KUKA KRL program: EPS_2_251524_MH2A_A_20251127083654.src

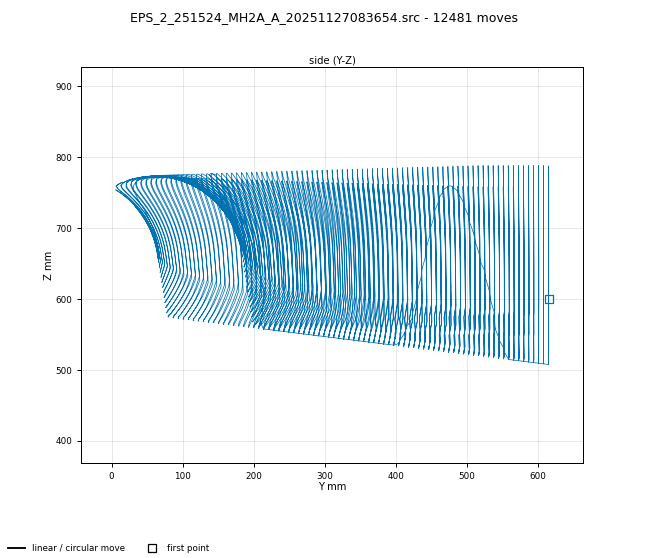
[picture p0: tool path of EPS_2_251524_MH2A_A_20251127083654.src, 12481 of 12483 moves have a stored position in this frame; points joined in program order, loops and branches not executed]
&ACCESS RVP
&REL 4
&COMMENT QRS 19112012
&PARAM EDITMASK = *
DEF PART()
EXT BAS (BAS_COMMAND :IN,REAL :IN )
INT I
BAS (#INITMOV,0 )

;KUKA QRS Post kuka4.cps  Date:22-06-2017 !

File_ID=2930

QRS_PRE_INIT()

;Init var - Until changes are made in qrs_pre_init
Outlet_Square_prg=0
Inlet_1_Square_prg=0
Inlet_2_Square_prg=0
Inlet_3_Square_prg=0
Inlet_4_Square_prg=0
Inlet_5_Square_prg=0

Outlet_1={X 0.000, Y 519.160, Z 687.500, B 0.000, E1 0.000 }
Inlet_1={X 0.000, Y 521.300, Z 657.500, B 0.000, E1 140.000 }
Outlet_1_type=201
Inlet_1_type=201
;QRS#1=Sidecore dimensions
;QRS#2=200-8" PVC SDR 35
;QRS#3=200-8" PVC SDR 35
;QRS#4=
;QRS#5=
;QRS#6=
;QRS#7=
;QRS#8=
;QRS#9=12-08 PSX
;QRS#10=12-08 PSX
;QRS#11=
;QRS#12=
;QRS#13=
;QRS#14=
;QRS#15=
;QRS#16=1220x127x1067 3,5'
;QRS#17=EPS Height
;QRS#18=788
;QRS#19=*
;QRS#20= UPDATED VERSION 22-06-2017
;QRS#21=*
Outlet_Square=0100
Inlet_1_Square=0100
Inlet_2_Square=0
Inlet_3_Square=0
Inlet_4_Square=0
Inlet_5_Square=0
Mill_Square=1
Outlet_Square_Prg=204
Inlet_1_Square_prg=204

QRS_INIT()

$ADVANCE=5

; T1
PTP {E1 173.595,E2 173.595}
PTP {X 0,Y 615.504,A -85,B 0,C 180,E1 173.595,E2 173.595,E3 0,E4 0,E5 0,E6 0}
QRS_SPEED_INIT()
LIN {X 0,Y 615.504,Z 600,A -85,B 0,C 180,E1 173.595,E2 173.595,E3 0,E4 0,E5 0,E6 0} C_VEL
LIN {X 0,Y 615.504,Z 517.862,A -85,B 0,C 180,E1 173.595,E2 173.595} C_VEL
LIN {X 0,Y 615.504,Z 509.682,A -85,B 0,C 180,E1 173.595,E2 173.595} C_VEL
LIN {X 0,Y 615.489,Z 507.682,A -85,B 0,C 180,E1 173.409,E2 173.409} C_VEL
LIN {X 0,Y 615.481,Z 507.697,A -85,B 0,C 180,E1 170.801,E2 170.801} C_VEL
LIN {X 0,Y 615.479,Z 507.69,A -85,B 0,C 180,E1 168.139,E2 168.139} C_VEL
LIN {X 0,Y 615.488,Z 507.682,A -85,B 0,C 180,E1 165.451,E2 165.451} C_VEL
LIN {X 0,Y 615.483,Z 507.699,A -85,B 0,C 180,E1 162.73,E2 162.73} C_VEL
LIN {X 0,Y 615.477,Z 507.687,A -85,B 0,C 180,E1 159.967,E2 159.967} C_VEL
LIN {X 0,Y 615.481,Z 507.683,A -85,B 0,C 180,E1 157.652,E2 157.652} C_VEL
LIN {X 0,Y 615.479,Z 507.692,A -85,B 0,C 180,E1 155.008,E2 155.008} C_VEL
LIN {X 0,Y 615.482,Z 507.688,A -85,B 0,C 180,E1 152.085,E2 152.085} C_VEL
LIN {X 0,Y 615.491,Z 507.714,A -85,B 0,C 180,E1 149.212,E2 149.212} C_VEL
LIN {X 0,Y 615.495,Z 524.435,A -85,B 0,C 180,E1 146.462,E2 146.462} C_VEL
LIN {X 0,Y 615.481,Z 542.244,A -85,B 0,C 180,E1 143.575,E2 143.575} C_VEL
LIN {X 0,Y 615.483,Z 546.958,A -85,B 0,C 180,E1 142.815,E2 142.815} C_VEL
LIN {X 0,Y 615.482,Z 654.02,A -85,B 0,C 180,E1 141.541,E2 141.541} C_VEL
LIN {X 0,Y 615.488,Z 667.054,A -85,B 0,C 180,E1 141.254,E2 141.254} C_VEL
LIN {X 0,Y 615.48,Z 679.367,A -85,B 0,C 180,E1 140.851,E2 140.851} C_VEL
LIN {X 0,Y 615.498,Z 691.041,A -85,B 0,C 180,E1 140.337,E2 140.337} C_VEL
LIN {X 0,Y 615.483,Z 702.98,A -85,B 0,C 180,E1 139.652,E2 139.652} C_VEL
LIN {X 0,Y 615.496,Z 713.375,A -85,B 0,C 180,E1 138.903,E2 138.903} C_VEL
LIN {X 0,Y 615.499,Z 722.741,A -85,B 0,C 180,E1 138.071,E2 138.071} C_VEL
LIN {X 0,Y 615.496,Z 731.335,A -85,B 0,C 180,E1 137.125,E2 137.125} C_VEL
LIN {X 0,Y 615.495,Z 738.265,A -85,B 0,C 180,E1 136.19,E2 136.19} C_VEL
LIN {X 0,Y 615.496,Z 744.904,A -85,B 0,C 180,E1 135.066,E2 135.066} C_VEL
LIN {X 0,Y 615.495,Z 749.711,A -85,B 0,C 180,E1 133.999,E2 133.999} C_VEL
LIN {X 0,Y 615.495,Z 752.959,A -85,B 0,C 180,E1 133.049,E2 133.049} C_VEL
LIN {X 0,Y 615.498,Z 755.309,A -85,B 0,C 180,E1 132.082,E2 132.082} C_VEL
LIN {X 0,Y 615.492,Z 756.779,A -85,B 0,C 180,E1 131.096,E2 131.096} C_VEL
LIN {X 0,Y 615.493,Z 757.346,A -85,B 0,C 180,E1 129.748,E2 129.748} C_VEL
LIN {X 0,Y 615.493,Z 756.882,A -85,B 0,C 180,E1 128.902,E2 128.902} C_VEL
LIN {X 0,Y 615.495,Z 755.644,A -85,B 0,C 180,E1 128.014,E2 128.014} C_VEL
LIN {X 0,Y 615.497,Z 753.167,A -85,B 0,C 180,E1 126.938,E2 126.938} C_VEL
LIN {X 0,Y 615.496,Z 749.426,A -85,B 0,C 180,E1 125.835,E2 125.835} C_VEL
LIN {X 0,Y 615.496,Z 744.143,A -85,B 0,C 180,E1 124.703,E2 124.703} C_VEL
LIN {X 0,Y 615.496,Z 737.021,A -85,B 0,C 180,E1 123.536,E2 123.536} C_VEL
LIN {X 0,Y 615.498,Z 730.229,A -85,B 0,C 180,E1 122.65,E2 122.65} C_VEL
LIN {X 0,Y 615.497,Z 722.8,A -85,B 0,C 180,E1 121.845,E2 121.845} C_VEL
LIN {X 0,Y 615.496,Z 713.317,A -85,B 0,C 180,E1 121.003,E2 121.003} C_VEL
LIN {X 0,Y 615.495,Z 702.902,A -85,B 0,C 180,E1 120.253,E2 120.253} C_VEL
LIN {X 0,Y 615.48,Z 691.58,A -85,B 0,C 180,E1 119.6,E2 119.6} C_VEL
LIN {X 0,Y 615.493,Z 679.846,A -85,B 0,C 180,E1 119.077,E2 119.077} C_VEL
LIN {X 0,Y 615.477,Z 667.095,A -85,B 0,C 180,E1 118.657,E2 118.657} C_VEL
LIN {X 0,Y 615.484,Z 654.766,A -85,B 0,C 180,E1 118.383,E2 118.383} C_VEL
LIN {X 0,Y 615.485,Z 578.99,A -85,B 0,C 180,E1 117.475,E2 117.475} C_VEL
LIN {X 0,Y 615.492,Z 546.957,A -85,B 0,C 180,E1 117.095,E2 117.095} C_VEL
LIN {X 0,Y 615.487,Z 529.495,A -85,B 0,C 180,E1 114.271,E2 114.271} C_VEL
LIN {X 0,Y 615.491,Z 512.144,A -85,B 0,C 180,E1 111.431,E2 111.431} C_VEL
LIN {X 0,Y 615.477,Z 507.687,A -85,B 0,C 180,E1 110.686,E2 110.686} C_VEL
LIN {X 0,Y 615.488,Z 507.683,A -85,B 0,C 180,E1 107.956,E2 107.956} C_VEL
LIN {X 0,Y 615.493,Z 507.701,A -85,B 0,C 180,E1 105.225,E2 105.225} C_VEL
LIN {X 0,Y 615.477,Z 507.686,A -85,B 0,C 180,E1 102.529,E2 102.529} C_VEL
LIN {X 0,Y 615.487,Z 507.684,A -85,B 0,C 180,E1 99.861,E2 99.861} C_VEL
LIN {X 0,Y 615.491,Z 507.7,A -85,B 0,C 180,E1 97.215,E2 97.215} C_VEL
LIN {X 0,Y 615.477,Z 507.688,A -85,B 0,C 180,E1 94.584,E2 94.584} C_VEL
LIN {X 0,Y 615.496,Z 507.68,A -85,B 0,C 180,E1 91.962,E2 91.962} C_VEL
LIN {X 0,Y 615.483,Z 507.694,A -85,B 0,C 180,E1 89.345,E2 89.345} C_VEL
LIN {X 0,Y 615.482,Z 507.693,A -85,B 0,C 180,E1 86.726,E2 86.726} C_VEL
LIN {X 0,Y 615.488,Z 507.681,A -85,B 0,C 180,E1 84.101,E2 84.101} C_VEL
LIN {X 0,Y 615.476,Z 507.69,A -85,B 0,C 180,E1 81.462,E2 81.462} C_VEL
LIN {X 0,Y 615.489,Z 507.696,A -85,B 0,C 180,E1 78.806,E2 78.806} C_VEL
LIN {X 0,Y 615.484,Z 507.682,A -85,B 0,C 180,E1 76.067,E2 76.067} C_VEL
LIN {X 0,Y 615.477,Z 507.689,A -85,B 0,C 180,E1 73.412,E2 73.412} C_VEL
LIN {X 0,Y 615.484,Z 507.695,A -85,B 0,C 180,E1 70.661,E2 70.661} C_VEL
LIN {X 0,Y 615.494,Z 507.68,A -85,B 0,C 180,E1 67.863,E2 67.863} C_VEL
LIN {X 0,Y 615.488,Z 507.696,A -85,B 0,C 180,E1 65.007,E2 65.007} C_VEL
LIN {X 0,Y 615.484,Z 507.684,A -85,B 0,C 180,E1 62.084,E2 62.084} C_VEL
LIN {X 0,Y 615.499,Z 507.679,A -85,B 0,C 180,E1 59.84,E2 59.84} C_VEL
LIN {X 0,Y 615.481,Z 507.684,A -85,B 0,C 180,E1 57.541,E2 57.541} C_VEL
LIN {X 0,Y 615.478,Z 507.69,A -85,B 0,C 180,E1 55.184,E2 55.184} C_VEL
LIN {X 0,Y 615.493,Z 507.699,A -85,B 0,C 180,E1 52.757,E2 52.757} C_VEL
LIN {X 0,Y 615.49,Z 507.682,A -85,B 0,C 180,E1 49.91,E2 49.91} C_VEL
LIN {X 0,Y 615.49,Z 507.681,A -85,B 0,C 180,E1 47.646,E2 47.646} C_VEL
LIN {X 0,Y 615.482,Z 507.693,A -85,B 0,C 180,E1 44.93,E2 44.93} C_VEL
LIN {X 0,Y 615.482,Z 507.688,A -85,B 0,C 180,E1 42.079,E2 42.079} C_VEL
LIN {X 0,Y 615.498,Z 507.68,A -85,B 0,C 180,E1 39.749,E2 39.749} C_VEL
LIN {X 0,Y 615.48,Z 507.691,A -85,B 0,C 180,E1 36.935,E2 36.935} C_VEL
LIN {X 0,Y 615.494,Z 507.695,A -85,B 0,C 180,E1 34.7,E2 34.7} C_VEL
LIN {X 0,Y 615.487,Z 507.682,A -85,B 0,C 180,E1 31.685,E2 31.685} C_VEL
LIN {X 0,Y 615.482,Z 507.683,A -85,B 0,C 180,E1 29.406,E2 29.406} C_VEL
LIN {X 0,Y 615.478,Z 507.687,A -85,B 0,C 180,E1 27.042,E2 27.042} C_VEL
LIN {X 0,Y 615.491,Z 507.696,A -85,B 0,C 180,E1 24.271,E2 24.271} C_VEL
LIN {X 0,Y 615.486,Z 507.682,A -85,B 0,C 180,E1 21.432,E2 21.432} C_VEL
LIN {X 0,Y 615.492,Z 507.693,A -85,B 0,C 180,E1 18.604,E2 18.604} C_VEL
LIN {X 0,Y 615.487,Z 507.689,A -85,B 0,C 180,E1 15.905,E2 15.905} C_VEL
LIN {X 0,Y 615.478,Z 507.684,A -85,B 0,C 180,E1 13.201,E2 13.201} C_VEL
LIN {X 0,Y 615.488,Z 507.693,A -85,B 0,C 180,E1 10.527,E2 10.527} C_VEL
LIN {X 0,Y 615.488,Z 507.69,A -85,B 0,C 180,E1 7.875,E2 7.875} C_VEL
LIN {X 0,Y 615.481,Z 507.683,A -85,B 0,C 180,E1 5.241,E2 5.241} C_VEL
LIN {X 0,Y 615.491,Z 507.688,A -85,B 0,C 180,E1 2.618,E2 2.618} C_VEL
LIN {X 0,Y 615.492,Z 507.695,A -85,B 0,C 180,E1 0,E2 0} C_VEL
LIN {X 0,Y 615.491,Z 507.682,A -85,B 0,C 180,E1 -2.618,E2 -2.618} C_VEL
LIN {X 0,Y 615.481,Z 507.686,A -85,B 0,C 180,E1 -5.242,E2 -5.242} C_VEL
LIN {X 0,Y 615.487,Z 507.702,A -85,B 0,C 180,E1 -7.876,E2 -7.876} C_VEL
LIN {X 0,Y 615.491,Z 507.684,A -85,B 0,C 180,E1 -10.527,E2 -10.527} C_VEL
LIN {X 0,Y 615.478,Z 507.685,A -85,B 0,C 180,E1 -13.202,E2 -13.202} C_VEL
LIN {X 0,Y 615.492,Z 507.699,A -85,B 0,C 180,E1 -15.905,E2 -15.905} C_VEL
LIN {X 0,Y 615.49,Z 507.684,A -85,B 0,C 180,E1 -18.646,E2 -18.646} C_VEL
LIN {X 0,Y 615.486,Z 507.685,A -85,B 0,C 180,E1 -21.432,E2 -21.432} C_VEL
LIN {X 0,Y 615.493,Z 507.694,A -85,B 0,C 180,E1 -24.272,E2 -24.272} C_VEL
LIN {X 0,Y 615.478,Z 507.684,A -85,B 0,C 180,E1 -27.042,E2 -27.042} C_VEL
LIN {X 0,Y 615.488,Z 507.691,A -85,B 0,C 180,E1 -29.794,E2 -29.794} C_VEL
LIN {X 0,Y 615.494,Z 507.691,A -85,B 0,C 180,E1 -32.457,E2 -32.457} C_VEL
LIN {X 0,Y 615.49,Z 507.684,A -85,B 0,C 180,E1 -34.815,E2 -34.815} C_VEL
LIN {X 0,Y 615.474,Z 507.684,A -85,B 0,C 180,E1 -37.243,E2 -37.243} C_VEL
LIN {X 0,Y 615.482,Z 507.698,A -85,B 0,C 180,E1 -40.088,E2 -40.088} C_VEL
LIN {X 0,Y 615.496,Z 507.697,A -85,B 0,C 180,E1 -42.353,E2 -42.353} C_VEL
LIN {X 0,Y 615.48,Z 507.684,A -85,B 0,C 180,E1 -45.07,E2 -45.07} C_VEL
LIN {X 0,Y 615.488,Z 507.689,A -85,B 0,C 180,E1 -47.92,E2 -47.92} C_VEL
LIN {X 0,Y 615.49,Z 507.699,A -85,B 0,C 180,E1 -50.249,E2 -50.249} C_VEL
LIN {X 0,Y 615.482,Z 507.685,A -85,B 0,C 180,E1 -53.065,E2 -53.065} C_VEL
LIN {X 0,Y 615.477,Z 507.684,A -85,B 0,C 180,E1 -55.301,E2 -55.301} C_VEL
LIN {X 0,Y 615.488,Z 507.683,A -85,B 0,C 180,E1 -57.67,E2 -57.67} C_VEL
LIN {X 0,Y 615.495,Z 507.695,A -85,B 0,C 180,E1 -60.593,E2 -60.593} C_VEL
LIN {X 0,Y 615.491,Z 507.686,A -85,B 0,C 180,E1 -62.955,E2 -62.955} C_VEL
LIN {X 0,Y 615.487,Z 507.683,A -85,B 0,C 180,E1 -65.727,E2 -65.727} C_VEL
LIN {X 0,Y 615.492,Z 507.756,A -85,B 0,C 180,E1 -67.837,E2 -67.837} C_VEL
LIN {X 0,Y 615.483,Z 528.07,A -85,B 0,C 180,E1 -70.661,E2 -70.661} C_VEL
LIN {X 0,Y 615.477,Z 548.18,A -85,B 0,C 180,E1 -73.412,E2 -73.412} C_VEL
LIN {X 0,Y 615.487,Z 568.265,A -85,B 0,C 180,E1 -76.125,E2 -76.125} C_VEL
LIN {X 0,Y 615.485,Z 576.034,A -85,B 0,C 180,E1 -77.134,E2 -77.134} C_VEL
LIN {X 0,Y 615.477,Z 683.784,A -85,B 0,C 180,E1 -78.41,E2 -78.41} C_VEL
LIN {X 0,Y 615.482,Z 696.314,A -85,B 0,C 180,E1 -78.681,E2 -78.681} C_VEL
LIN {X 0,Y 615.497,Z 709.493,A -85,B 0,C 180,E1 -79.109,E2 -79.109} C_VEL
LIN {X 0,Y 615.48,Z 721.461,A -85,B 0,C 180,E1 -79.638,E2 -79.638} C_VEL
LIN {X 0,Y 615.481,Z 732.983,A -85,B 0,C 180,E1 -80.303,E2 -80.303} C_VEL
LIN {X 0,Y 615.499,Z 743.33,A -85,B 0,C 180,E1 -81.049,E2 -81.049} C_VEL
LIN {X 0,Y 615.497,Z 751.802,A -85,B 0,C 180,E1 -81.793,E2 -81.793} C_VEL
LIN {X 0,Y 615.498,Z 759.599,A -85,B 0,C 180,E1 -82.619,E2 -82.619} C_VEL
LIN {X 0,Y 615.496,Z 767.197,A -85,B 0,C 180,E1 -83.607,E2 -83.607} C_VEL
LIN {X 0,Y 615.498,Z 774.2,A -85,B 0,C 180,E1 -84.758,E2 -84.758} C_VEL
LIN {X 0,Y 615.493,Z 778.848,A -85,B 0,C 180,E1 -85.743,E2 -85.743} C_VEL
LIN {X 0,Y 615.495,Z 782.396,A -85,B 0,C 180,E1 -86.726,E2 -86.726} C_VEL
LIN {X 0,Y 615.497,Z 784.231,A -85,B 0,C 180,E1 -87.381,E2 -87.381} C_VEL
LIN {X 0,Y 615.496,Z 785.607,A -85,B 0,C 180,E1 -88.036,E2 -88.036} C_VEL
LIN {X 0,Y 615.496,Z 787.173,A -85,B 0,C 180,E1 -89.345,E2 -89.345} C_VEL
LIN {X 0,Y 615.494,Z 787.389,A -85,B 0,C 180,E1 -89.999,E2 -89.999} C_VEL
LIN {X 0,Y 615.496,Z 786.581,A -85,B 0,C 180,E1 -91.308,E2 -91.308} C_VEL
LIN {X 0,Y 615.496,Z 785.61,A -85,B 0,C 180,E1 -91.962,E2 -91.962} C_VEL
LIN {X 0,Y 615.497,Z 784.235,A -85,B 0,C 180,E1 -92.617,E2 -92.617} C_VEL
LIN {X 0,Y 615.496,Z 781.353,A -85,B 0,C 180,E1 -93.6,E2 -93.6} C_VEL
LIN {X 0,Y 615.498,Z 777.446,A -85,B 0,C 180,E1 -94.583,E2 -94.583} C_VEL
LIN {X 0,Y 615.499,Z 772.41,A -85,B 0,C 180,E1 -95.569,E2 -95.569} C_VEL
LIN {X 0,Y 615.496,Z 765.87,A -85,B 0,C 180,E1 -96.583,E2 -96.583} C_VEL
LIN {X 0,Y 615.497,Z 758.142,A -85,B 0,C 180,E1 -97.544,E2 -97.544} C_VEL
LIN {X 0,Y 615.498,Z 750.056,A -85,B 0,C 180,E1 -98.37,E2 -98.37} C_VEL
LIN {X 0,Y 615.499,Z 740.181,A -85,B 0,C 180,E1 -99.198,E2 -99.198} C_VEL
LIN {X 0,Y 615.483,Z 729,A -85,B 0,C 180,E1 -99.944,E2 -99.944} C_VEL
LIN {X 0,Y 615.481,Z 718.045,A -85,B 0,C 180,E1 -100.526,E2 -100.526} C_VEL
LIN {X 0,Y 615.499,Z 705.435,A -85,B 0,C 180,E1 -101.042,E2 -101.042} C_VEL
LIN {X 0,Y 615.479,Z 693.112,A -85,B 0,C 180,E1 -101.401,E2 -101.401} C_VEL
LIN {X 0,Y 615.477,Z 679.544,A -85,B 0,C 180,E1 -101.651,E2 -101.651} C_VEL
LIN {X 0,Y 615.486,Z 575.649,A -85,B 0,C 180,E1 -102.885,E2 -102.885} C_VEL
LIN {X 0,Y 615.479,Z 554.474,A -85,B 0,C 180,E1 -105.734,E2 -105.734} C_VEL
LIN {X 0,Y 615.479,Z 534.611,A -85,B 0,C 180,E1 -108.44,E2 -108.44} C_VEL
LIN {X 0,Y 615.497,Z 514.247,A -85,B 0,C 180,E1 -111.255,E2 -111.255} C_VEL
LIN {X 0,Y 615.489,Z 507.683,A -85,B 0,C 180,E1 -112.187,E2 -112.187} C_VEL
LIN {X 0,Y 615.488,Z 507.687,A -85,B 0,C 180,E1 -114.99,E2 -114.99} C_VEL
LIN {X 0,Y 615.483,Z 507.69,A -85,B 0,C 180,E1 -117.914,E2 -117.914} C_VEL
LIN {X 0,Y 615.499,Z 507.681,A -85,B 0,C 180,E1 -120.158,E2 -120.158} C_VEL
LIN {X 0,Y 615.481,Z 507.683,A -85,B 0,C 180,E1 -122.456,E2 -122.456} C_VEL
LIN {X 0,Y 615.478,Z 507.687,A -85,B 0,C 180,E1 -124.814,E2 -124.814} C_VEL
LIN {X 0,Y 615.496,Z 507.693,A -85,B 0,C 180,E1 -127.24,E2 -127.24} C_VEL
LIN {X 0,Y 615.49,Z 507.684,A -85,B 0,C 180,E1 -130.089,E2 -130.089} C_VEL
LIN {X 0,Y 615.49,Z 507.681,A -85,B 0,C 180,E1 -132.351,E2 -132.351} C_VEL
LIN {X 0,Y 615.481,Z 507.691,A -85,B 0,C 180,E1 -135.067,E2 -135.067} C_VEL
LIN {X 0,Y 615.477,Z 507.69,A -85,B 0,C 180,E1 -137.919,E2 -137.919} C_VEL
LIN {X 0,Y 615.498,Z 507.68,A -85,B 0,C 180,E1 -140.25,E2 -140.25} C_VEL
LIN {X 0,Y 615.48,Z 507.691,A -85,B 0,C 180,E1 -143.062,E2 -143.062} C_VEL
LIN {X 0,Y 615.494,Z 507.696,A -85,B 0,C 180,E1 -145.296,E2 -145.296} C_VEL
LIN {X 0,Y 615.485,Z 507.683,A -85,B 0,C 180,E1 -148.314,E2 -148.314} C_VEL
LIN {X 0,Y 615.482,Z 507.683,A -85,B 0,C 180,E1 -150.593,E2 -150.593} C_VEL
LIN {X 0,Y 615.478,Z 507.69,A -85,B 0,C 180,E1 -152.954,E2 -152.954} C_VEL
LIN {X 0,Y 615.478,Z 507.695,A -85,B 0,C 180,E1 -155.727,E2 -155.727} C_VEL
LIN {X 0,Y 615.486,Z 507.683,A -85,B 0,C 180,E1 -158.568,E2 -158.568} C_VEL
LIN {X 0,Y 615.494,Z 507.7,A -85,B 0,C 180,E1 -161.389,E2 -161.389} C_VEL
LIN {X 0,Y 615.48,Z 507.686,A -85,B 0,C 180,E1 -164.094,E2 -164.094} C_VEL
LIN {X 0,Y 615.478,Z 507.687,A -85,B 0,C 180,E1 -166.798,E2 -166.798} C_VEL
LIN {X 0,Y 615.488,Z 507.701,A -85,B 0,C 180,E1 -169.473,E2 -169.473} C_VEL
LIN {X 0,Y 615.479,Z 507.686,A -85,B 0,C 180,E1 -172.124,E2 -172.124} C_VEL
LIN {X 0,Y 615.481,Z 507.686,A -85,B 0,C 180,E1 -174.758,E2 -174.758} C_VEL
LIN {X 0,Y 615.495,Z 507.7,A -85,B 0,C 180,E1 -177.382,E2 -177.382} C_VEL
LIN {X 0,Y 615.477,Z 507.688,A -85,B 0,C 180,E1 -180,E2 -180} C_VEL
LIN {X 0,Y 615.492,Z 507.682,A -85,B 0,C 180,E1 -182.617,E2 -182.617} C_VEL
LIN {X 0,Y 615.481,Z 507.698,A -85,B 0,C 180,E1 -185.241,E2 -185.241} C_VEL
LIN {X 0,Y 615.489,Z 507.682,A -85,B 0,C 180,E1 -186.591,E2 -186.591} C_VEL
LIN {X 0,Y 614.808,Z 507.844,A -85,B 0,C 180,E1 -187.137,E2 -187.137} C_VEL
LIN {X 0,Y 611.969,Z 508.251,A -85,B 0,C 180,E1 -188.023,E2 -188.023} C_VEL
LIN {X 0,Y 609.577,Z 508.566,A -85,B 0,C 180,E1 -188.735,E2 -188.735} C_VEL
LIN {X 0,Y 608.541,Z 508.686,A -85,B 0,C 180,E1 -189.285,E2 -189.285} C_VEL
LIN {X 0,Y 608.452,Z 508.694,A -85,B 0,C 180,E1 -189.471,E2 -189.471} C_VEL
LIN {X 0,Y 608.456,Z 508.688,A -85,B 0,C 180,E1 -192,E2 -192} C_VEL
LIN {X 0,Y 608.473,Z 508.686,A -85,B 0,C 180,E1 -194.72,E2 -194.72} C_VEL
LIN {X 0,Y 608.447,Z 508.698,A -85,B 0,C 180,E1 -197.476,E2 -197.476} C_VEL
LIN {X 0,Y 608.457,Z 508.687,A -85,B 0,C 180,E1 -200.274,E2 -200.274} C_VEL
LIN {X 0,Y 608.449,Z 508.688,A -85,B 0,C 180,E1 -202.478,E2 -202.478} C_VEL
LIN {X 0,Y 608.451,Z 508.697,A -85,B 0,C 180,E1 -205.301,E2 -205.301} C_VEL
LIN {X 0,Y 608.444,Z 508.697,A -85,B 0,C 180,E1 -207.518,E2 -207.518} C_VEL
LIN {X 0,Y 608.451,Z 508.69,A -85,B 0,C 180,E1 -209.972,E2 -209.972} C_VEL
LIN {X 0,Y 608.513,Z 508.816,A -85,B 0,C 180,E1 -210.734,E2 -210.734} C_VEL
LIN {X 0,Y 608.493,Z 526.519,A -85,B 0,C 180,E1 -213.668,E2 -213.668} C_VEL
LIN {X 0,Y 608.482,Z 543.856,A -85,B 0,C 180,E1 -216.5,E2 -216.5} C_VEL
LIN {X 0,Y 608.461,Z 547.129,A -85,B 0,C 180,E1 -217.03,E2 -217.03} C_VEL
LIN {X 0,Y 608.555,Z 654.443,A -85,B 0,C 180,E1 -218.331,E2 -218.331} C_VEL
LIN {X 0,Y 608.526,Z 667.914,A -85,B 0,C 180,E1 -218.636,E2 -218.636} C_VEL
LIN {X 0,Y 608.529,Z 680.513,A -85,B 0,C 180,E1 -219.061,E2 -219.061} C_VEL
LIN {X 0,Y 608.52,Z 692.231,A -85,B 0,C 180,E1 -219.596,E2 -219.596} C_VEL
LIN {X 0,Y 608.485,Z 704.174,A -85,B 0,C 180,E1 -220.3,E2 -220.3} C_VEL
LIN {X 0,Y 608.486,Z 714.511,A -85,B 0,C 180,E1 -221.064,E2 -221.064} C_VEL
LIN {X 0,Y 608.458,Z 723.364,A -85,B 0,C 180,E1 -221.867,E2 -221.867} C_VEL
LIN {X 0,Y 608.466,Z 731.678,A -85,B 0,C 180,E1 -222.788,E2 -222.788} C_VEL
LIN {X 0,Y 608.438,Z 739.591,A -85,B 0,C 180,E1 -223.872,E2 -223.872} C_VEL
LIN {X 0,Y 608.455,Z 746.008,A -85,B 0,C 180,E1 -225.002,E2 -225.002} C_VEL
LIN {X 0,Y 608.43,Z 750.892,A -85,B 0,C 180,E1 -226.129,E2 -226.129} C_VEL
LIN {X 0,Y 608.433,Z 753.859,A -85,B 0,C 180,E1 -227.04,E2 -227.04} C_VEL
LIN {X 0,Y 608.426,Z 755.989,A -85,B 0,C 180,E1 -227.937,E2 -227.937} C_VEL
LIN {X 0,Y 608.429,Z 757.303,A -85,B 0,C 180,E1 -228.823,E2 -228.823} C_VEL
LIN {X 0,Y 608.441,Z 757.925,A -85,B 0,C 180,E1 -229.697,E2 -229.697} C_VEL
LIN {X 0,Y 608.42,Z 757.783,A -85,B 0,C 180,E1 -230.708,E2 -230.708} C_VEL
LIN {X 0,Y 608.417,Z 756.643,A -85,B 0,C 180,E1 -231.765,E2 -231.765} C_VEL
LIN {X 0,Y 608.432,Z 753.765,A -85,B 0,C 180,E1 -233.085,E2 -233.085} C_VEL
LIN {X 0,Y 608.447,Z 749.419,A -85,B 0,C 180,E1 -234.34,E2 -234.34} C_VEL
LIN {X 0,Y 608.429,Z 743.685,A -85,B 0,C 180,E1 -235.53,E2 -235.53} C_VEL
LIN {X 0,Y 608.44,Z 737.509,A -85,B 0,C 180,E1 -236.528,E2 -236.528} C_VEL
LIN {X 0,Y 608.47,Z 730.26,A -85,B 0,C 180,E1 -237.476,E2 -237.476} C_VEL
LIN {X 0,Y 608.46,Z 721.613,A -85,B 0,C 180,E1 -238.394,E2 -238.394} C_VEL
LIN {X 0,Y 608.49,Z 711.492,A -85,B 0,C 180,E1 -239.265,E2 -239.265} C_VEL
LIN {X 0,Y 608.487,Z 700.535,A -85,B 0,C 180,E1 -240.024,E2 -240.024} C_VEL
LIN {X 0,Y 608.503,Z 690.043,A -85,B 0,C 180,E1 -240.604,E2 -240.604} C_VEL
LIN {X 0,Y 608.518,Z 677.026,A -85,B 0,C 180,E1 -241.16,E2 -241.16} C_VEL
LIN {X 0,Y 608.521,Z 664.353,A -85,B 0,C 180,E1 -241.552,E2 -241.552} C_VEL
LIN {X 0,Y 608.548,Z 651.153,A -85,B 0,C 180,E1 -241.81,E2 -241.81} C_VEL
LIN {X 0,Y 608.458,Z 547.155,A -85,B 0,C 180,E1 -243.056,E2 -243.056} C_VEL
LIN {X 0,Y 608.482,Z 530.028,A -85,B 0,C 180,E1 -245.846,E2 -245.846} C_VEL
LIN {X 0,Y 608.51,Z 512.946,A -85,B 0,C 180,E1 -248.667,E2 -248.667} C_VEL
LIN {X 0,Y 608.469,Z 508.687,A -85,B 0,C 180,E1 -249.411,E2 -249.411} C_VEL
LIN {X 0,Y 608.447,Z 508.688,A -85,B 0,C 180,E1 -251.829,E2 -251.829} C_VEL
LIN {X 0,Y 608.476,Z 508.692,A -85,B 0,C 180,E1 -254.595,E2 -254.595} C_VEL
LIN {X 0,Y 608.471,Z 508.687,A -85,B 0,C 180,E1 -257.324,E2 -257.324} C_VEL
LIN {X 0,Y 608.455,Z 508.687,A -85,B 0,C 180,E1 -260.024,E2 -260.024} C_VEL
LIN {X 0,Y 608.485,Z 508.691,A -85,B 0,C 180,E1 -262.702,E2 -262.702} C_VEL
LIN {X 0,Y 608.447,Z 508.691,A -85,B 0,C 180,E1 -265.363,E2 -265.363} C_VEL
LIN {X 0,Y 608.466,Z 508.685,A -85,B 0,C 180,E1 -268.015,E2 -268.015} C_VEL
LIN {X 0,Y 608.478,Z 508.69,A -85,B 0,C 180,E1 -270.663,E2 -270.663} C_VEL
LIN {X 0,Y 608.476,Z 508.689,A -85,B 0,C 180,E1 -273.312,E2 -273.312} C_VEL
LIN {X 0,Y 608.483,Z 508.683,A -85,B 0,C 180,E1 -275.968,E2 -275.968} C_VEL
LIN {X 0,Y 608.449,Z 508.692,A -85,B 0,C 180,E1 -278.637,E2 -278.637} C_VEL
LIN {X 0,Y 608.478,Z 508.689,A -85,B 0,C 180,E1 -281.325,E2 -281.325} C_VEL
LIN {X 0,Y 608.468,Z 508.685,A -85,B 0,C 180,E1 -284.038,E2 -284.038} C_VEL
LIN {X 0,Y 608.454,Z 508.692,A -85,B 0,C 180,E1 -286.785,E2 -286.785} C_VEL
LIN {X 0,Y 608.452,Z 508.69,A -85,B 0,C 180,E1 -289.571,E2 -289.571} C_VEL
LIN {X 0,Y 608.459,Z 508.687,A -85,B 0,C 180,E1 -292.477,E2 -292.477} C_VEL
LIN {X 0,Y 608.455,Z 508.688,A -85,B 0,C 180,E1 -294.572,E2 -294.572} C_VEL
LIN {X 0,Y 608.482,Z 508.695,A -85,B 0,C 180,E1 -297.209,E2 -297.209} C_VEL
LIN {X 0,Y 608.468,Z 508.686,A -85,B 0,C 180,E1 -299.972,E2 -299.972} C_VEL
LIN {X 0,Y 608.458,Z 508.687,A -85,B 0,C 180,E1 -302.523,E2 -302.523} C_VEL
LIN {X 0,Y 608.438,Z 508.7,A -85,B 0,C 180,E1 -305.279,E2 -305.279} C_VEL
LIN {X 0,Y 608.472,Z 508.688,A -85,B 0,C 180,E1 -307.747,E2 -307.747} C_VEL
LIN {X 0,Y 608.451,Z 508.687,A -85,B 0,C 180,E1 -310.329,E2 -310.329} C_VEL
LIN {X 0,Y 608.486,Z 508.693,A -85,B 0,C 180,E1 -313.311,E2 -313.311} C_VEL
LIN {X 0,Y 608.469,Z 508.685,A -85,B 0,C 180,E1 -316.131,E2 -316.131} C_VEL
LIN {X 0,Y 608.449,Z 508.689,A -85,B 0,C 180,E1 -318.823,E2 -318.823} C_VEL
LIN {X 0,Y 608.468,Z 508.696,A -85,B 0,C 180,E1 -321.412,E2 -321.412} C_VEL
LIN {X 0,Y 608.449,Z 508.69,A -85,B 0,C 180,E1 -323.955,E2 -323.955} C_VEL
LIN {X 0,Y 608.469,Z 508.685,A -85,B 0,C 180,E1 -326.33,E2 -326.33} C_VEL
LIN {X 0,Y 608.447,Z 508.688,A -85,B 0,C 180,E1 -328.733,E2 -328.733} C_VEL
LIN {X 0,Y 608.48,Z 508.692,A -85,B 0,C 180,E1 -331.38,E2 -331.38} C_VEL
LIN {X 0,Y 608.479,Z 508.684,A -85,B 0,C 180,E1 -334.279,E2 -334.279} C_VEL
LIN {X 0,Y 608.449,Z 508.688,A -85,B 0,C 180,E1 -336.876,E2 -336.876} C_VEL
LIN {X 0,Y 608.469,Z 508.691,A -85,B 0,C 180,E1 -339.323,E2 -339.323} C_VEL
LIN {X 0,Y 608.452,Z 508.695,A -85,B 0,C 180,E1 -341.829,E2 -341.829} C_VEL
LIN {X 0,Y 608.467,Z 508.685,A -85,B 0,C 180,E1 -344.594,E2 -344.594} C_VEL
LIN {X 0,Y 608.48,Z 508.688,A -85,B 0,C 180,E1 -347.324,E2 -347.324} C_VEL
LIN {X 0,Y 608.458,Z 508.692,A -85,B 0,C 180,E1 -350.023,E2 -350.023} C_VEL
LIN {X 0,Y 608.462,Z 508.686,A -85,B 0,C 180,E1 -352.701,E2 -352.701} C_VEL
LIN {X 0,Y 608.463,Z 508.689,A -85,B 0,C 180,E1 -355.363,E2 -355.363} C_VEL
LIN {X 0,Y 608.46,Z 508.693,A -85,B 0,C 180,E1 -358.015,E2 -358.015} C_VEL
LIN {X 0,Y 608.48,Z 508.684,A -85,B 0,C 180,E1 -360.662,E2 -360.662} C_VEL
LIN {X 0,Y 608.477,Z 508.686,A -85,B 0,C 180,E1 -363.311,E2 -363.311} C_VEL
LIN {X 0,Y 608.472,Z 508.694,A -85,B 0,C 180,E1 -365.967,E2 -365.967} C_VEL
LIN {X 0,Y 608.46,Z 508.687,A -85,B 0,C 180,E1 -368.636,E2 -368.636} C_VEL
LIN {X 0,Y 608.446,Z 508.689,A -85,B 0,C 180,E1 -371.325,E2 -371.325} C_VEL
LIN {X 0,Y 608.477,Z 508.694,A -85,B 0,C 180,E1 -374.038,E2 -374.038} C_VEL
LIN {X 0,Y 608.478,Z 508.684,A -85,B 0,C 180,E1 -376.784,E2 -376.784} C_VEL
LIN {X 0,Y 608.451,Z 508.69,A -85,B 0,C 180,E1 -379.571,E2 -379.571} C_VEL
LIN {X 0,Y 608.466,Z 508.689,A -85,B 0,C 180,E1 -382.476,E2 -382.476} C_VEL
LIN {X 0,Y 608.455,Z 508.689,A -85,B 0,C 180,E1 -384.571,E2 -384.571} C_VEL
LIN {X 0,Y 608.473,Z 508.684,A -85,B 0,C 180,E1 -387.205,E2 -387.205} C_VEL
LIN {X 0,Y 608.473,Z 508.692,A -85,B 0,C 180,E1 -389.971,E2 -389.971} C_VEL
LIN {X 0,Y 608.457,Z 508.687,A -85,B 0,C 180,E1 -392.88,E2 -392.88} C_VEL
LIN {X 0,Y 608.449,Z 508.687,A -85,B 0,C 180,E1 -395.278,E2 -395.278} C_VEL
LIN {X 0,Y 608.471,Z 508.696,A -85,B 0,C 180,E1 -398.24,E2 -398.24} C_VEL
LIN {X 0,Y 608.457,Z 508.686,A -85,B 0,C 180,E1 -401.341,E2 -401.341} C_VEL
LIN {X 0,Y 608.455,Z 508.698,A -85,B 0,C 180,E1 -404.263,E2 -404.263} C_VEL
LIN {X 0,Y 608.453,Z 508.687,A -85,B 0,C 180,E1 -407.039,E2 -407.039} C_VEL
LIN {X 0,Y 608.459,Z 508.687,A -85,B 0,C 180,E1 -409.696,E2 -409.696} C_VEL
LIN {X 0,Y 608.473,Z 508.694,A -85,B 0,C 180,E1 -412.253,E2 -412.253} C_VEL
LIN {X 0,Y 608.446,Z 508.689,A -85,B 0,C 180,E1 -415.095,E2 -415.095} C_VEL
LIN {X 0,Y 608.459,Z 508.686,A -85,B 0,C 180,E1 -417.479,E2 -417.479} C_VEL
LIN {X 0,Y 608.464,Z 508.693,A -85,B 0,C 180,E1 -420.219,E2 -420.219} C_VEL
LIN {X 0,Y 608.485,Z 508.688,A -85,B 0,C 180,E1 -422.792,E2 -422.792} C_VEL
LIN {X 0,Y 608.456,Z 508.687,A -85,B 0,C 180,E1 -425.428,E2 -425.428} C_VEL
LIN {X 0,Y 608.488,Z 508.885,A -85,B 0,C 180,E1 -427.729,E2 -427.729} C_VEL
LIN {X 0,Y 608.545,Z 525.571,A -85,B 0,C 180,E1 -430.08,E2 -430.08} C_VEL
LIN {X 0,Y 608.525,Z 545.72,A -85,B 0,C 180,E1 -432.871,E2 -432.871} C_VEL
LIN {X 0,Y 608.481,Z 567.128,A -85,B 0,C 180,E1 -435.791,E2 -435.791} C_VEL
LIN {X 0,Y 608.489,Z 576.069,A -85,B 0,C 180,E1 -436.983,E2 -436.983} C_VEL
LIN {X 0,Y 608.535,Z 683.899,A -85,B 0,C 180,E1 -438.276,E2 -438.276} C_VEL
LIN {X 0,Y 608.534,Z 697.185,A -85,B 0,C 180,E1 -438.571,E2 -438.571} C_VEL
LIN {X 0,Y 608.541,Z 710.38,A -85,B 0,C 180,E1 -439.011,E2 -439.011} C_VEL
LIN {X 0,Y 608.498,Z 721.618,A -85,B 0,C 180,E1 -439.518,E2 -439.518} C_VEL
LIN {X 0,Y 608.471,Z 733.184,A -85,B 0,C 180,E1 -440.19,E2 -440.19} C_VEL
LIN {X 0,Y 608.485,Z 743.582,A -85,B 0,C 180,E1 -440.945,E2 -440.945} C_VEL
LIN {X 0,Y 608.475,Z 752.102,A -85,B 0,C 180,E1 -441.698,E2 -441.698} C_VEL
LIN {X 0,Y 608.471,Z 759.953,A -85,B 0,C 180,E1 -442.533,E2 -442.533} C_VEL
LIN {X 0,Y 608.461,Z 767.284,A -85,B 0,C 180,E1 -443.484,E2 -443.484} C_VEL
LIN {X 0,Y 608.45,Z 772.861,A -85,B 0,C 180,E1 -444.365,E2 -444.365} C_VEL
LIN {X 0,Y 608.432,Z 777.946,A -85,B 0,C 180,E1 -445.361,E2 -445.361} C_VEL
LIN {X 0,Y 608.449,Z 781.893,A -85,B 0,C 180,E1 -446.357,E2 -446.357} C_VEL
LIN {X 0,Y 608.425,Z 784.807,A -85,B 0,C 180,E1 -447.351,E2 -447.351} C_VEL
LIN {X 0,Y 608.442,Z 786.2,A -85,B 0,C 180,E1 -448.013,E2 -448.013} C_VEL
LIN {X 0,Y 608.439,Z 787.783,A -85,B 0,C 180,E1 -449.337,E2 -449.337} C_VEL
LIN {X 0,Y 608.434,Z 788,A -85,B 0,C 180,E1 -449.999,E2 -449.999} C_VEL
LIN {X 0,Y 608.448,Z 787.185,A -85,B 0,C 180,E1 -451.323,E2 -451.323} C_VEL
LIN {X 0,Y 608.441,Z 786.203,A -85,B 0,C 180,E1 -451.985,E2 -451.985} C_VEL
LIN {X 0,Y 608.425,Z 784.812,A -85,B 0,C 180,E1 -452.647,E2 -452.647} C_VEL
LIN {X 0,Y 608.449,Z 781.899,A -85,B 0,C 180,E1 -453.641,E2 -453.641} C_VEL
LIN {X 0,Y 608.432,Z 777.954,A -85,B 0,C 180,E1 -454.637,E2 -454.637} C_VEL
LIN {X 0,Y 608.437,Z 771.883,A -85,B 0,C 180,E1 -455.8,E2 -455.8} C_VEL
LIN {X 0,Y 608.461,Z 765.242,A -85,B 0,C 180,E1 -456.798,E2 -456.798} C_VEL
LIN {X 0,Y 608.455,Z 756.998,A -85,B 0,C 180,E1 -457.799,E2 -457.799} C_VEL
LIN {X 0,Y 608.472,Z 748.548,A -85,B 0,C 180,E1 -458.635,E2 -458.635} C_VEL
LIN {X 0,Y 608.474,Z 738.105,A -85,B 0,C 180,E1 -459.472,E2 -459.472} C_VEL
LIN {X 0,Y 608.482,Z 727.773,A -85,B 0,C 180,E1 -460.144,E2 -460.144} C_VEL
LIN {X 0,Y 608.521,Z 716.258,A -85,B 0,C 180,E1 -460.74,E2 -460.74} C_VEL
LIN {X 0,Y 608.528,Z 704.901,A -85,B 0,C 180,E1 -461.192,E2 -461.192} C_VEL
LIN {X 0,Y 608.546,Z 691.398,A -85,B 0,C 180,E1 -461.575,E2 -461.575} C_VEL
LIN {X 0,Y 608.543,Z 678.165,A -85,B 0,C 180,E1 -461.807,E2 -461.807} C_VEL
LIN {X 0,Y 608.525,Z 576.233,A -85,B 0,C 180,E1 -463.014,E2 -463.014} C_VEL
LIN {X 0,Y 608.489,Z 574.698,A -85,B 0,C 180,E1 -463.185,E2 -463.185} C_VEL
LIN {X 0,Y 608.489,Z 553.29,A -85,B 0,C 180,E1 -466.092,E2 -466.092} C_VEL
LIN {X 0,Y 608.511,Z 534.153,A -85,B 0,C 180,E1 -468.726,E2 -468.726} C_VEL
LIN {X 0,Y 608.573,Z 514.251,A -85,B 0,C 180,E1 -471.509,E2 -471.509} C_VEL
LIN {X 0,Y 608.455,Z 508.689,A -85,B 0,C 180,E1 -472.315,E2 -472.315} C_VEL
LIN {X 0,Y 608.455,Z 508.687,A -85,B 0,C 180,E1 -474.57,E2 -474.57} C_VEL
LIN {X 0,Y 608.484,Z 508.689,A -85,B 0,C 180,E1 -477.208,E2 -477.208} C_VEL
LIN {X 0,Y 608.467,Z 508.688,A -85,B 0,C 180,E1 -479.971,E2 -479.971} C_VEL
LIN {X 0,Y 608.457,Z 508.687,A -85,B 0,C 180,E1 -482.521,E2 -482.521} C_VEL
LIN {X 0,Y 608.443,Z 508.69,A -85,B 0,C 180,E1 -484.904,E2 -484.904} C_VEL
LIN {X 0,Y 608.471,Z 508.691,A -85,B 0,C 180,E1 -487.745,E2 -487.745} C_VEL
LIN {X 0,Y 608.45,Z 508.688,A -85,B 0,C 180,E1 -490.328,E2 -490.328} C_VEL
LIN {X 0,Y 608.485,Z 508.691,A -85,B 0,C 180,E1 -493.31,E2 -493.31} C_VEL
LIN {X 0,Y 608.466,Z 508.687,A -85,B 0,C 180,E1 -496.13,E2 -496.13} C_VEL
LIN {X 0,Y 608.449,Z 508.689,A -85,B 0,C 180,E1 -498.823,E2 -498.823} C_VEL
LIN {X 0,Y 608.465,Z 508.696,A -85,B 0,C 180,E1 -501.411,E2 -501.411} C_VEL
LIN {X 0,Y 608.472,Z 508.688,A -85,B 0,C 180,E1 -503.949,E2 -503.949} C_VEL
LIN {X 0,Y 608.462,Z 508.686,A -85,B 0,C 180,E1 -506.329,E2 -506.329} C_VEL
LIN {X 0,Y 608.469,Z 508.686,A -85,B 0,C 180,E1 -508.726,E2 -508.726} C_VEL
LIN {X 0,Y 608.471,Z 508.695,A -85,B 0,C 180,E1 -511.378,E2 -511.378} C_VEL
LIN {X 0,Y 608.475,Z 508.684,A -85,B 0,C 180,E1 -514.275,E2 -514.275} C_VEL
LIN {X 0,Y 608.447,Z 508.69,A -85,B 0,C 180,E1 -516.876,E2 -516.876} C_VEL
LIN {X 0,Y 608.465,Z 508.695,A -85,B 0,C 180,E1 -519.318,E2 -519.318} C_VEL
LIN {X 0,Y 608.447,Z 508.692,A -85,B 0,C 180,E1 -521.828,E2 -521.828} C_VEL
LIN {X 0,Y 608.463,Z 508.686,A -85,B 0,C 180,E1 -524.594,E2 -524.594} C_VEL
LIN {X 0,Y 608.475,Z 508.693,A -85,B 0,C 180,E1 -527.323,E2 -527.323} C_VEL
LIN {X 0,Y 608.449,Z 508.689,A -85,B 0,C 180,E1 -530.022,E2 -530.022} C_VEL
LIN {X 0,Y 608.474,Z 508.685,A -85,B 0,C 180,E1 -532.7,E2 -532.7} C_VEL
LIN {X 0,Y 608.466,Z 508.696,A -85,B 0,C 180,E1 -535.362,E2 -535.362} C_VEL
LIN {X 0,Y 608.446,Z 508.69,A -85,B 0,C 180,E1 -538.014,E2 -538.014} C_VEL
LIN {X 0,Y 608.478,Z 508.685,A -85,B 0,C 180,E1 -540.661,E2 -540.661} C_VEL
LIN {X 0,Y 608.477,Z 508.693,A -85,B 0,C 180,E1 -543.31,E2 -543.31} C_VEL
LIN {X 0,Y 608.453,Z 508.689,A -85,B 0,C 180,E1 -545.967,E2 -545.967} C_VEL
LIN {X 0,Y 608.457,Z 508.687,A -85,B 0,C 180,E1 -548.636,E2 -548.636} C_VEL
LIN {X 0,Y 608.452,Z 508.694,A -85,B 0,C 180,E1 -549.471,E2 -549.471} C_VEL
LIN {X 0,Y 607.772,Z 508.774,A -85,B 0,C 180,E1 -550.024,E2 -550.024} C_VEL
LIN {X 0,Y 604.917,Z 509.131,A -85,B 0,C 180,E1 -550.921,E2 -550.921} C_VEL
LIN {X 0,Y 602.515,Z 509.433,A -85,B 0,C 180,E1 -551.642,E2 -551.642} C_VEL
LIN {X 0,Y 601.488,Z 509.556,A -85,B 0,C 180,E1 -552.199,E2 -552.199} C_VEL
LIN {X 0,Y 601.405,Z 509.565,A -85,B 0,C 180,E1 -552.388,E2 -552.388} C_VEL
LIN {X 0,Y 601.426,Z 509.565,A -85,B 0,C 180,E1 -554.897,E2 -554.897} C_VEL
LIN {X 0,Y 601.426,Z 509.567,A -85,B 0,C 180,E1 -556.986,E2 -556.986} C_VEL
LIN {X 0,Y 601.401,Z 509.57,A -85,B 0,C 180,E1 -559.809,E2 -559.809} C_VEL
LIN {X 0,Y 601.405,Z 509.566,A -85,B 0,C 180,E1 -562.606,E2 -562.606} C_VEL
LIN {X 0,Y 601.397,Z 509.569,A -85,B 0,C 180,E1 -564.878,E2 -564.878} C_VEL
LIN {X 0,Y 601.416,Z 509.567,A -85,B 0,C 180,E1 -567.867,E2 -567.867} C_VEL
LIN {X 0,Y 601.462,Z 509.691,A -85,B 0,C 180,E1 -570.647,E2 -570.647} C_VEL
LIN {X 0,Y 601.485,Z 525.543,A -85,B 0,C 180,E1 -573.309,E2 -573.309} C_VEL
LIN {X 0,Y 601.435,Z 541.842,A -85,B 0,C 180,E1 -576.007,E2 -576.007} C_VEL
LIN {X 0,Y 601.41,Z 547.095,A -85,B 0,C 180,E1 -576.869,E2 -576.869} C_VEL
LIN {X 0,Y 601.667,Z 551.434,A -85,B 0,C 180,E1 -576.942,E2 -576.942} C_VEL
LIN {X 0,Y 601.599,Z 654.123,A -85,B 0,C 180,E1 -578.187,E2 -578.187} C_VEL
LIN {X 0,Y 601.589,Z 667.528,A -85,B 0,C 180,E1 -578.492,E2 -578.492} C_VEL
LIN {X 0,Y 601.549,Z 680.309,A -85,B 0,C 180,E1 -578.924,E2 -578.924} C_VEL
LIN {X 0,Y 601.516,Z 691.806,A -85,B 0,C 180,E1 -579.45,E2 -579.45} C_VEL
LIN {X 0,Y 601.468,Z 702.829,A -85,B 0,C 180,E1 -580.096,E2 -580.096} C_VEL
LIN {X 0,Y 601.462,Z 713.421,A -85,B 0,C 180,E1 -580.87,E2 -580.87} C_VEL
LIN {X 0,Y 601.408,Z 723.323,A -85,B 0,C 180,E1 -581.766,E2 -581.766} C_VEL
LIN {X 0,Y 601.379,Z 731.443,A -85,B 0,C 180,E1 -582.673,E2 -582.673} C_VEL
LIN {X 0,Y 601.375,Z 738.208,A -85,B 0,C 180,E1 -583.59,E2 -583.59} C_VEL
LIN {X 0,Y 601.369,Z 745.096,A -85,B 0,C 180,E1 -584.758,E2 -584.758} C_VEL
LIN {X 0,Y 601.355,Z 750.387,A -85,B 0,C 180,E1 -585.945,E2 -585.945} C_VEL
LIN {X 0,Y 601.335,Z 753.532,A -85,B 0,C 180,E1 -586.882,E2 -586.882} C_VEL
LIN {X 0,Y 601.338,Z 754.931,A -85,B 0,C 180,E1 -587.416,E2 -587.416} C_VEL
LIN {X 0,Y 601.322,Z 756.827,A -85,B 0,C 180,E1 -588.417,E2 -588.417} C_VEL
LIN {X 0,Y 601.311,Z 757.827,A -85,B 0,C 180,E1 -589.438,E2 -589.438} C_VEL
LIN {X 0,Y 601.315,Z 757.906,A -85,B 0,C 180,E1 -590.478,E2 -590.478} C_VEL
LIN {X 0,Y 601.329,Z 756.739,A -85,B 0,C 180,E1 -591.727,E2 -591.727} C_VEL
LIN {X 0,Y 601.346,Z 754.02,A -85,B 0,C 180,E1 -593.024,E2 -593.024} C_VEL
LIN {X 0,Y 601.348,Z 750.02,A -85,B 0,C 180,E1 -594.244,E2 -594.244} C_VEL
LIN {X 0,Y 601.35,Z 744.344,A -85,B 0,C 180,E1 -595.473,E2 -595.473} C_VEL
LIN {X 0,Y 601.358,Z 738.002,A -85,B 0,C 180,E1 -596.531,E2 -596.531} C_VEL
LIN {X 0,Y 601.403,Z 730.904,A -85,B 0,C 180,E1 -597.484,E2 -597.484} C_VEL
LIN {X 0,Y 601.401,Z 722.178,A -85,B 0,C 180,E1 -598.439,E2 -598.439} C_VEL
LIN {X 0,Y 601.453,Z 711.753,A -85,B 0,C 180,E1 -599.354,E2 -599.354} C_VEL
LIN {X 0,Y 601.479,Z 700.734,A -85,B 0,C 180,E1 -600.13,E2 -600.13} C_VEL
LIN {X 0,Y 601.518,Z 689.011,A -85,B 0,C 180,E1 -600.779,E2 -600.779} C_VEL
LIN {X 0,Y 601.549,Z 676.074,A -85,B 0,C 180,E1 -601.327,E2 -601.327} C_VEL
LIN {X 0,Y 601.56,Z 663.185,A -85,B 0,C 180,E1 -601.714,E2 -601.714} C_VEL
LIN {X 0,Y 601.601,Z 649.907,A -85,B 0,C 180,E1 -601.965,E2 -601.965} C_VEL
LIN {X 0,Y 601.647,Z 548.669,A -85,B 0,C 180,E1 -603.181,E2 -603.181} C_VEL
LIN {X 0,Y 601.41,Z 547.119,A -85,B 0,C 180,E1 -603.217,E2 -603.217} C_VEL
LIN {X 0,Y 601.459,Z 531.077,A -85,B 0,C 180,E1 -605.861,E2 -605.861} C_VEL
LIN {X 0,Y 601.515,Z 514.758,A -85,B 0,C 180,E1 -608.586,E2 -608.586} C_VEL
LIN {X 0,Y 601.427,Z 509.565,A -85,B 0,C 180,E1 -609.479,E2 -609.479} C_VEL
LIN {X 0,Y 601.401,Z 509.57,A -85,B 0,C 180,E1 -612.313,E2 -612.313} C_VEL
LIN {X 0,Y 601.418,Z 509.568,A -85,B 0,C 180,E1 -614.41,E2 -614.41} C_VEL
LIN {X 0,Y 601.419,Z 509.567,A -85,B 0,C 180,E1 -617.173,E2 -617.173} C_VEL
LIN {X 0,Y 601.431,Z 509.561,A -85,B 0,C 180,E1 -619.906,E2 -619.906} C_VEL
LIN {X 0,Y 601.453,Z 509.566,A -85,B 0,C 180,E1 -622.616,E2 -622.616} C_VEL
LIN {X 0,Y 601.416,Z 509.567,A -85,B 0,C 180,E1 -625.309,E2 -625.309} C_VEL
LIN {X 0,Y 601.434,Z 509.561,A -85,B 0,C 180,E1 -627.992,E2 -627.992} C_VEL
LIN {X 0,Y 601.449,Z 509.566,A -85,B 0,C 180,E1 -630.67,E2 -630.67} C_VEL
LIN {X 0,Y 601.427,Z 509.566,A -85,B 0,C 180,E1 -633.35,E2 -633.35} C_VEL
LIN {X 0,Y 601.432,Z 509.561,A -85,B 0,C 180,E1 -636.038,E2 -636.038} C_VEL
LIN {X 0,Y 601.41,Z 509.57,A -85,B 0,C 180,E1 -638.739,E2 -638.739} C_VEL
LIN {X 0,Y 601.435,Z 509.565,A -85,B 0,C 180,E1 -641.459,E2 -641.459} C_VEL
LIN {X 0,Y 601.418,Z 509.563,A -85,B 0,C 180,E1 -644.206,E2 -644.206} C_VEL
LIN {X 0,Y 601.421,Z 509.572,A -85,B 0,C 180,E1 -646.987,E2 -646.987} C_VEL
LIN {X 0,Y 601.406,Z 509.566,A -85,B 0,C 180,E1 -649.81,E2 -649.81} C_VEL
LIN {X 0,Y 601.412,Z 509.567,A -85,B 0,C 180,E1 -652.684,E2 -652.684} C_VEL
LIN {X 0,Y 601.402,Z 509.571,A -85,B 0,C 180,E1 -654.879,E2 -654.879} C_VEL
LIN {X 0,Y 601.419,Z 509.571,A -85,B 0,C 180,E1 -657.364,E2 -657.364} C_VEL
LIN {X 0,Y 601.429,Z 509.562,A -85,B 0,C 180,E1 -660.165,E2 -660.165} C_VEL
LIN {X 0,Y 601.42,Z 509.565,A -85,B 0,C 180,E1 -662.716,E2 -662.716} C_VEL
LIN {X 0,Y 601.393,Z 509.574,A -85,B 0,C 180,E1 -665.112,E2 -665.112} C_VEL
LIN {X 0,Y 601.438,Z 509.57,A -85,B 0,C 180,E1 -667.42,E2 -667.42} C_VEL
LIN {X 0,Y 601.412,Z 509.565,A -85,B 0,C 180,E1 -669.996,E2 -669.996} C_VEL
LIN {X 0,Y 601.414,Z 509.565,A -85,B 0,C 180,E1 -672.671,E2 -672.671} C_VEL
LIN {X 0,Y 601.429,Z 509.571,A -85,B 0,C 180,E1 -675.483,E2 -675.483} C_VEL
LIN {X 0,Y 601.422,Z 509.563,A -85,B 0,C 180,E1 -678.408,E2 -678.408} C_VEL
LIN {X 0,Y 601.435,Z 509.563,A -85,B 0,C 180,E1 -680.876,E2 -680.876} C_VEL
LIN {X 0,Y 601.402,Z 509.576,A -85,B 0,C 180,E1 -683.417,E2 -683.417} C_VEL
LIN {X 0,Y 601.436,Z 509.563,A -85,B 0,C 180,E1 -686.065,E2 -686.065} C_VEL
LIN {X 0,Y 601.422,Z 509.563,A -85,B 0,C 180,E1 -688.546,E2 -688.546} C_VEL
LIN {X 0,Y 601.439,Z 509.568,A -85,B 0,C 180,E1 -691.374,E2 -691.374} C_VEL
LIN {X 0,Y 601.42,Z 509.565,A -85,B 0,C 180,E1 -694.133,E2 -694.133} C_VEL
LIN {X 0,Y 601.399,Z 509.565,A -85,B 0,C 180,E1 -696.589,E2 -696.589} C_VEL
LIN {X 0,Y 601.433,Z 509.57,A -85,B 0,C 180,E1 -699.479,E2 -699.479} C_VEL
LIN {X 0,Y 601.396,Z 509.567,A -85,B 0,C 180,E1 -702.312,E2 -702.312} C_VEL
LIN {X 0,Y 601.413,Z 509.564,A -85,B 0,C 180,E1 -704.409,E2 -704.409} C_VEL
LIN {X 0,Y 601.423,Z 509.565,A -85,B 0,C 180,E1 -707.172,E2 -707.172} C_VEL
LIN {X 0,Y 601.435,Z 509.569,A -85,B 0,C 180,E1 -709.905,E2 -709.905} C_VEL
LIN {X 0,Y 601.442,Z 509.56,A -85,B 0,C 180,E1 -712.615,E2 -712.615} C_VEL
LIN {X 0,Y 601.43,Z 509.565,A -85,B 0,C 180,E1 -715.308,E2 -715.308} C_VEL
LIN {X 0,Y 601.43,Z 509.569,A -85,B 0,C 180,E1 -717.991,E2 -717.991} C_VEL
LIN {X 0,Y 601.452,Z 509.559,A -85,B 0,C 180,E1 -720.67,E2 -720.67} C_VEL
LIN {X 0,Y 601.428,Z 509.565,A -85,B 0,C 180,E1 -723.35,E2 -723.35} C_VEL
LIN {X 0,Y 601.425,Z 509.571,A -85,B 0,C 180,E1 -726.037,E2 -726.037} C_VEL
LIN {X 0,Y 601.419,Z 509.563,A -85,B 0,C 180,E1 -728.738,E2 -728.738} C_VEL
LIN {X 0,Y 601.42,Z 509.566,A -85,B 0,C 180,E1 -731.459,E2 -731.459} C_VEL
LIN {X 0,Y 601.427,Z 509.569,A -85,B 0,C 180,E1 -734.206,E2 -734.206} C_VEL
LIN {X 0,Y 601.435,Z 509.561,A -85,B 0,C 180,E1 -736.986,E2 -736.986} C_VEL
LIN {X 0,Y 601.408,Z 509.571,A -85,B 0,C 180,E1 -739.81,E2 -739.81} C_VEL
LIN {X 0,Y 601.418,Z 509.565,A -85,B 0,C 180,E1 -742.683,E2 -742.683} C_VEL
LIN {X 0,Y 601.404,Z 509.565,A -85,B 0,C 180,E1 -744.879,E2 -744.879} C_VEL
LIN {X 0,Y 601.414,Z 509.564,A -85,B 0,C 180,E1 -747.361,E2 -747.361} C_VEL
LIN {X 0,Y 601.436,Z 509.572,A -85,B 0,C 180,E1 -750.164,E2 -750.164} C_VEL
LIN {X 0,Y 601.426,Z 509.564,A -85,B 0,C 180,E1 -752.715,E2 -752.715} C_VEL
LIN {X 0,Y 601.417,Z 509.563,A -85,B 0,C 180,E1 -755.114,E2 -755.114} C_VEL
LIN {X 0,Y 601.438,Z 509.561,A -85,B 0,C 180,E1 -757.419,E2 -757.419} C_VEL
LIN {X 0,Y 601.409,Z 509.571,A -85,B 0,C 180,E1 -759.996,E2 -759.996} C_VEL
LIN {X 0,Y 601.416,Z 509.567,A -85,B 0,C 180,E1 -762.67,E2 -762.67} C_VEL
LIN {X 0,Y 601.405,Z 509.565,A -85,B 0,C 180,E1 -765.479,E2 -765.479} C_VEL
LIN {X 0,Y 601.418,Z 509.563,A -85,B 0,C 180,E1 -767.409,E2 -767.409} C_VEL
LIN {X 0,Y 601.409,Z 509.569,A -85,B 0,C 180,E1 -770.004,E2 -770.004} C_VEL
LIN {X 0,Y 601.442,Z 509.566,A -85,B 0,C 180,E1 -772.618,E2 -772.618} C_VEL
LIN {X 0,Y 601.409,Z 509.565,A -85,B 0,C 180,E1 -775.067,E2 -775.067} C_VEL
LIN {X 0,Y 601.429,Z 509.562,A -85,B 0,C 180,E1 -777.483,E2 -777.483} C_VEL
LIN {X 0,Y 601.435,Z 509.563,A -85,B 0,C 180,E1 -779.851,E2 -779.851} C_VEL
LIN {X 0,Y 601.422,Z 509.571,A -85,B 0,C 180,E1 -782.637,E2 -782.637} C_VEL
LIN {X 0,Y 601.407,Z 509.567,A -85,B 0,C 180,E1 -785.121,E2 -785.121} C_VEL
LIN {X 0,Y 601.472,Z 509.759,A -85,B 0,C 180,E1 -787.58,E2 -787.58} C_VEL
LIN {X 0,Y 601.606,Z 520.764,A -85,B 0,C 180,E1 -789.159,E2 -789.159} C_VEL
LIN {X 0,Y 601.558,Z 540.682,A -85,B 0,C 180,E1 -791.964,E2 -791.964} C_VEL
LIN {X 0,Y 601.492,Z 560.831,A -85,B 0,C 180,E1 -794.757,E2 -794.757} C_VEL
LIN {X 0,Y 601.466,Z 576.069,A -85,B 0,C 180,E1 -796.828,E2 -796.828} C_VEL
LIN {X 0,Y 601.655,Z 602.9,A -85,B 0,C 180,E1 -797.155,E2 -797.155} C_VEL
LIN {X 0,Y 601.604,Z 683.899,A -85,B 0,C 180,E1 -798.138,E2 -798.138} C_VEL
LIN {X 0,Y 601.573,Z 697.185,A -85,B 0,C 180,E1 -798.437,E2 -798.437} C_VEL
LIN {X 0,Y 601.551,Z 708.905,A -85,B 0,C 180,E1 -798.825,E2 -798.825} C_VEL
LIN {X 0,Y 601.515,Z 719.905,A -85,B 0,C 180,E1 -799.31,E2 -799.31} C_VEL
LIN {X 0,Y 601.466,Z 730.565,A -85,B 0,C 180,E1 -799.905,E2 -799.905} C_VEL
LIN {X 0,Y 601.446,Z 741.464,A -85,B 0,C 180,E1 -800.668,E2 -800.668} C_VEL
LIN {X 0,Y 601.429,Z 752.102,A -85,B 0,C 180,E1 -801.6,E2 -801.6} C_VEL
LIN {X 0,Y 601.418,Z 759.953,A -85,B 0,C 180,E1 -802.445,E2 -802.445} C_VEL
LIN {X 0,Y 601.371,Z 767.221,A -85,B 0,C 180,E1 -803.397,E2 -803.397} C_VEL
LIN {X 0,Y 601.372,Z 772.861,A -85,B 0,C 180,E1 -804.298,E2 -804.298} C_VEL
LIN {X 0,Y 601.337,Z 777.946,A -85,B 0,C 180,E1 -805.306,E2 -805.306} C_VEL
LIN {X 0,Y 601.367,Z 781.893,A -85,B 0,C 180,E1 -806.314,E2 -806.314} C_VEL
LIN {X 0,Y 601.325,Z 784.807,A -85,B 0,C 180,E1 -807.32,E2 -807.32} C_VEL
LIN {X 0,Y 601.34,Z 786.2,A -85,B 0,C 180,E1 -807.99,E2 -807.99} C_VEL
LIN {X 0,Y 601.339,Z 787.783,A -85,B 0,C 180,E1 -809.329,E2 -809.329} C_VEL
LIN {X 0,Y 601.335,Z 788,A -85,B 0,C 180,E1 -809.999,E2 -809.999} C_VEL
LIN {X 0,Y 601.348,Z 787.185,A -85,B 0,C 180,E1 -811.338,E2 -811.338} C_VEL
LIN {X 0,Y 601.34,Z 786.203,A -85,B 0,C 180,E1 -812.008,E2 -812.008} C_VEL
LIN {X 0,Y 601.325,Z 784.812,A -85,B 0,C 180,E1 -812.679,E2 -812.679} C_VEL
LIN {X 0,Y 601.367,Z 781.899,A -85,B 0,C 180,E1 -813.684,E2 -813.684} C_VEL
LIN {X 0,Y 601.337,Z 777.954,A -85,B 0,C 180,E1 -814.692,E2 -814.692} C_VEL
LIN {X 0,Y 601.372,Z 771.883,A -85,B 0,C 180,E1 -815.868,E2 -815.868} C_VEL
LIN {X 0,Y 601.387,Z 765.243,A -85,B 0,C 180,E1 -816.879,E2 -816.879} C_VEL
LIN {X 0,Y 601.4,Z 756.998,A -85,B 0,C 180,E1 -817.891,E2 -817.891} C_VEL
LIN {X 0,Y 601.436,Z 748.548,A -85,B 0,C 180,E1 -818.737,E2 -818.737} C_VEL
LIN {X 0,Y 601.441,Z 738.106,A -85,B 0,C 180,E1 -819.584,E2 -819.584} C_VEL
LIN {X 0,Y 601.484,Z 727.774,A -85,B 0,C 180,E1 -820.263,E2 -820.263} C_VEL
LIN {X 0,Y 601.536,Z 716.913,A -85,B 0,C 180,E1 -820.835,E2 -820.835} C_VEL
LIN {X 0,Y 601.558,Z 704.403,A -85,B 0,C 180,E1 -821.34,E2 -821.34} C_VEL
LIN {X 0,Y 601.589,Z 691.398,A -85,B 0,C 180,E1 -821.71,E2 -821.71} C_VEL
LIN {X 0,Y 601.61,Z 678.165,A -85,B 0,C 180,E1 -821.945,E2 -821.945} C_VEL
LIN {X 0,Y 601.497,Z 576.233,A -85,B 0,C 180,E1 -823.169,E2 -823.169} C_VEL
LIN {X 0,Y 601.445,Z 574.698,A -85,B 0,C 180,E1 -823.342,E2 -823.342} C_VEL
LIN {X 0,Y 601.495,Z 554.549,A -85,B 0,C 180,E1 -826.11,E2 -826.11} C_VEL
LIN {X 0,Y 601.561,Z 536.504,A -85,B 0,C 180,E1 -828.621,E2 -828.621} C_VEL
LIN {X 0,Y 601.658,Z 515.51,A -85,B 0,C 180,E1 -831.588,E2 -831.588} C_VEL
LIN {X 0,Y 601.417,Z 509.568,A -85,B 0,C 180,E1 -832.46,E2 -832.46} C_VEL
LIN {X 0,Y 601.403,Z 509.568,A -85,B 0,C 180,E1 -834.877,E2 -834.877} C_VEL
LIN {X 0,Y 601.42,Z 509.568,A -85,B 0,C 180,E1 -837.866,E2 -837.866} C_VEL
LIN {X 0,Y 601.426,Z 509.564,A -85,B 0,C 180,E1 -840.163,E2 -840.163} C_VEL
LIN {X 0,Y 601.42,Z 509.564,A -85,B 0,C 180,E1 -842.715,E2 -842.715} C_VEL
LIN {X 0,Y 601.391,Z 509.571,A -85,B 0,C 180,E1 -845.111,E2 -845.111} C_VEL
LIN {X 0,Y 601.434,Z 509.572,A -85,B 0,C 180,E1 -847.418,E2 -847.418} C_VEL
LIN {X 0,Y 601.408,Z 509.567,A -85,B 0,C 180,E1 -849.994,E2 -849.994} C_VEL
LIN {X 0,Y 601.411,Z 509.565,A -85,B 0,C 180,E1 -852.669,E2 -852.669} C_VEL
LIN {X 0,Y 601.419,Z 509.574,A -85,B 0,C 180,E1 -855.481,E2 -855.481} C_VEL
LIN {X 0,Y 601.418,Z 509.563,A -85,B 0,C 180,E1 -858.406,E2 -858.406} C_VEL
LIN {X 0,Y 601.431,Z 509.564,A -85,B 0,C 180,E1 -860.875,E2 -860.875} C_VEL
LIN {X 0,Y 601.437,Z 509.567,A -85,B 0,C 180,E1 -863.733,E2 -863.733} C_VEL
LIN {X 0,Y 601.43,Z 509.564,A -85,B 0,C 180,E1 -866.062,E2 -866.062} C_VEL
LIN {X 0,Y 601.434,Z 509.561,A -85,B 0,C 180,E1 -868.541,E2 -868.541} C_VEL
LIN {X 0,Y 601.43,Z 509.572,A -85,B 0,C 180,E1 -871.373,E2 -871.373} C_VEL
LIN {X 0,Y 601.415,Z 509.565,A -85,B 0,C 180,E1 -874.129,E2 -874.129} C_VEL
LIN {X 0,Y 601.416,Z 509.564,A -85,B 0,C 180,E1 -876.589,E2 -876.589} C_VEL
LIN {X 0,Y 601.427,Z 509.572,A -85,B 0,C 180,E1 -879.478,E2 -879.478} C_VEL
LIN {X 0,Y 601.392,Z 509.567,A -85,B 0,C 180,E1 -882.311,E2 -882.311} C_VEL
LIN {X 0,Y 601.408,Z 509.564,A -85,B 0,C 180,E1 -884.408,E2 -884.408} C_VEL
LIN {X 0,Y 601.419,Z 509.57,A -85,B 0,C 180,E1 -887.171,E2 -887.171} C_VEL
LIN {X 0,Y 601.428,Z 509.565,A -85,B 0,C 180,E1 -889.905,E2 -889.905} C_VEL
LIN {X 0,Y 601.444,Z 509.56,A -85,B 0,C 180,E1 -892.615,E2 -892.615} C_VEL
LIN {X 0,Y 601.432,Z 509.571,A -85,B 0,C 180,E1 -895.308,E2 -895.308} C_VEL
LIN {X 0,Y 601.416,Z 509.565,A -85,B 0,C 180,E1 -897.991,E2 -897.991} C_VEL
LIN {X 0,Y 601.448,Z 509.56,A -85,B 0,C 180,E1 -900.669,E2 -900.669} C_VEL
LIN {X 0,Y 601.428,Z 509.572,A -85,B 0,C 180,E1 -903.349,E2 -903.349} C_VEL
LIN {X 0,Y 601.406,Z 509.567,A -85,B 0,C 180,E1 -906.037,E2 -906.037} C_VEL
LIN {X 0,Y 601.434,Z 509.563,A -85,B 0,C 180,E1 -908.737,E2 -908.737} C_VEL
LIN {X 0,Y 601.427,Z 509.573,A -85,B 0,C 180,E1 -911.458,E2 -911.458} C_VEL
LIN {X 0,Y 601.405,Z 509.565,A -85,B 0,C 180,E1 -912.388,E2 -912.388} C_VEL
LIN {X 0,Y 600.743,Z 509.652,A -85,B 0,C 180,E1 -912.947,E2 -912.947} C_VEL
LIN {X 0,Y 597.892,Z 510.006,A -85,B 0,C 180,E1 -913.855,E2 -913.855} C_VEL
LIN {X 0,Y 595.48,Z 510.308,A -85,B 0,C 180,E1 -914.585,E2 -914.585} C_VEL
LIN {X 0,Y 594.442,Z 510.439,A -85,B 0,C 180,E1 -915.148,E2 -915.148} C_VEL
LIN {X 0,Y 594.356,Z 510.447,A -85,B 0,C 180,E1 -915.339,E2 -915.339} C_VEL
LIN {X 0,Y 594.373,Z 510.444,A -85,B 0,C 180,E1 -917.904,E2 -917.904} C_VEL
LIN {X 0,Y 594.376,Z 510.444,A -85,B 0,C 180,E1 -920.919,E2 -920.919} C_VEL
LIN {X 0,Y 594.384,Z 510.445,A -85,B 0,C 180,E1 -923.704,E2 -923.704} C_VEL
LIN {X 0,Y 594.379,Z 510.442,A -85,B 0,C 180,E1 -926.699,E2 -926.699} C_VEL
LIN {X 0,Y 594.378,Z 510.446,A -85,B 0,C 180,E1 -928.998,E2 -928.998} C_VEL
LIN {X 0,Y 594.441,Z 510.551,A -85,B 0,C 180,E1 -930.556,E2 -930.556} C_VEL
LIN {X 0,Y 594.488,Z 523.31,A -85,B 0,C 180,E1 -932.729,E2 -932.729} C_VEL
LIN {X 0,Y 594.405,Z 540.494,A -85,B 0,C 180,E1 -935.613,E2 -935.613} C_VEL
LIN {X 0,Y 594.362,Z 547.185,A -85,B 0,C 180,E1 -936.725,E2 -936.725} C_VEL
LIN {X 0,Y 594.753,Z 551.448,A -85,B 0,C 180,E1 -936.787,E2 -936.787} C_VEL
LIN {X 0,Y 594.649,Z 654.549,A -85,B 0,C 180,E1 -938.055,E2 -938.055} C_VEL
LIN {X 0,Y 594.622,Z 667.947,A -85,B 0,C 180,E1 -938.366,E2 -938.366} C_VEL
LIN {X 0,Y 594.587,Z 680.229,A -85,B 0,C 180,E1 -938.789,E2 -938.789} C_VEL
LIN {X 0,Y 594.512,Z 692.098,A -85,B 0,C 180,E1 -939.34,E2 -939.34} C_VEL
LIN {X 0,Y 594.447,Z 703.786,A -85,B 0,C 180,E1 -940.041,E2 -940.041} C_VEL
LIN {X 0,Y 594.416,Z 714.261,A -85,B 0,C 180,E1 -940.828,E2 -940.828} C_VEL
LIN {X 0,Y 594.379,Z 723.212,A -85,B 0,C 180,E1 -941.656,E2 -941.656} C_VEL
LIN {X 0,Y 594.313,Z 731.677,A -85,B 0,C 180,E1 -942.614,E2 -942.614} C_VEL
LIN {X 0,Y 594.295,Z 738.561,A -85,B 0,C 180,E1 -943.567,E2 -943.567} C_VEL
LIN {X 0,Y 594.294,Z 744.192,A -85,B 0,C 180,E1 -944.524,E2 -944.524} C_VEL
LIN {X 0,Y 594.264,Z 748.7,A -85,B 0,C 180,E1 -945.475,E2 -945.475} C_VEL
LIN {X 0,Y 594.246,Z 753.073,A -85,B 0,C 180,E1 -946.691,E2 -946.691} C_VEL
LIN {X 0,Y 594.248,Z 755.422,A -85,B 0,C 180,E1 -947.616,E2 -947.616} C_VEL
LIN {X 0,Y 594.215,Z 756.994,A -85,B 0,C 180,E1 -948.524,E2 -948.524} C_VEL
LIN {X 0,Y 594.232,Z 757.822,A -85,B 0,C 180,E1 -949.423,E2 -949.423} C_VEL
LIN {X 0,Y 594.212,Z 757.946,A -85,B 0,C 180,E1 -950.308,E2 -950.308} C_VEL
LIN {X 0,Y 594.204,Z 757.28,A -85,B 0,C 180,E1 -951.317,E2 -951.317} C_VEL
LIN {X 0,Y 594.222,Z 755.553,A -85,B 0,C 180,E1 -952.412,E2 -952.412} C_VEL
LIN {X 0,Y 594.264,Z 751.974,A -85,B 0,C 180,E1 -953.751,E2 -953.751} C_VEL
LIN {X 0,Y 594.261,Z 746.759,A -85,B 0,C 180,E1 -955.052,E2 -955.052} C_VEL
LIN {X 0,Y 594.295,Z 740.396,A -85,B 0,C 180,E1 -956.235,E2 -956.235} C_VEL
LIN {X 0,Y 594.306,Z 733.268,A -85,B 0,C 180,E1 -957.275,E2 -957.275} C_VEL
LIN {X 0,Y 594.37,Z 724.684,A -85,B 0,C 180,E1 -958.28,E2 -958.28} C_VEL
LIN {X 0,Y 594.422,Z 715.58,A -85,B 0,C 180,E1 -959.149,E2 -959.149} C_VEL
LIN {X 0,Y 594.451,Z 705.079,A -85,B 0,C 180,E1 -959.962,E2 -959.962} C_VEL
LIN {X 0,Y 594.495,Z 694.459,A -85,B 0,C 180,E1 -960.621,E2 -960.621} C_VEL
LIN {X 0,Y 594.564,Z 682.505,A -85,B 0,C 180,E1 -961.206,E2 -961.206} C_VEL
LIN {X 0,Y 594.599,Z 670.729,A -85,B 0,C 180,E1 -961.642,E2 -961.642} C_VEL
LIN {X 0,Y 594.672,Z 657.949,A -85,B 0,C 180,E1 -961.97,E2 -961.97} C_VEL
LIN {X 0,Y 594.683,Z 642.828,A -85,B 0,C 180,E1 -962.196,E2 -962.196} C_VEL
LIN {X 0,Y 594.629,Z 548.848,A -85,B 0,C 180,E1 -963.337,E2 -963.337} C_VEL
LIN {X 0,Y 594.384,Z 546.999,A -85,B 0,C 180,E1 -963.395,E2 -963.395} C_VEL
LIN {X 0,Y 594.442,Z 530.71,A -85,B 0,C 180,E1 -966.114,E2 -966.114} C_VEL
LIN {X 0,Y 594.525,Z 513.39,A -85,B 0,C 180,E1 -969.046,E2 -969.046} C_VEL
LIN {X 0,Y 594.374,Z 510.445,A -85,B 0,C 180,E1 -969.586,E2 -969.586} C_VEL
LIN {X 0,Y 594.379,Z 510.442,A -85,B 0,C 180,E1 -972.097,E2 -972.097} C_VEL
LIN {X 0,Y 594.369,Z 510.444,A -85,B 0,C 180,E1 -974.22,E2 -974.22} C_VEL
LIN {X 0,Y 594.368,Z 510.448,A -85,B 0,C 180,E1 -977.018,E2 -977.018} C_VEL
LIN {X 0,Y 594.39,Z 510.439,A -85,B 0,C 180,E1 -979.785,E2 -979.785} C_VEL
LIN {X 0,Y 594.401,Z 510.443,A -85,B 0,C 180,E1 -982.528,E2 -982.528} C_VEL
LIN {X 0,Y 594.387,Z 510.443,A -85,B 0,C 180,E1 -985.253,E2 -985.253} C_VEL
LIN {X 0,Y 594.403,Z 510.437,A -85,B 0,C 180,E1 -987.968,E2 -987.968} C_VEL
LIN {X 0,Y 594.42,Z 510.441,A -85,B 0,C 180,E1 -990.678,E2 -990.678} C_VEL
LIN {X 0,Y 594.379,Z 510.444,A -85,B 0,C 180,E1 -993.39,E2 -993.39} C_VEL
LIN {X 0,Y 594.381,Z 510.44,A -85,B 0,C 180,E1 -996.11,E2 -996.11} C_VEL
LIN {X 0,Y 594.378,Z 510.448,A -85,B 0,C 180,E1 -998.843,E2 -998.843} C_VEL
LIN {X 0,Y 594.394,Z 510.44,A -85,B 0,C 180,E1 -1001.597,E2 -1001.597} C_VEL
LIN {X 0,Y 594.388,Z 510.44,A -85,B 0,C 180,E1 -1004.378,E2 -1004.378} C_VEL
LIN {X 0,Y 594.383,Z 510.449,A -85,B 0,C 180,E1 -1007.194,E2 -1007.194} C_VEL
LIN {X 0,Y 594.374,Z 510.441,A -85,B 0,C 180,E1 -1010.055,E2 -1010.055} C_VEL
LIN {X 0,Y 594.357,Z 510.45,A -85,B 0,C 180,E1 -1012.968,E2 -1012.968} C_VEL
LIN {X 0,Y 594.374,Z 510.452,A -85,B 0,C 180,E1 -1015.194,E2 -1015.194} C_VEL
LIN {X 0,Y 594.387,Z 510.444,A -85,B 0,C 180,E1 -1017.528,E2 -1017.528} C_VEL
LIN {X 0,Y 594.389,Z 510.439,A -85,B 0,C 180,E1 -1020.329,E2 -1020.329} C_VEL
LIN {X 0,Y 594.379,Z 510.445,A -85,B 0,C 180,E1 -1022.951,E2 -1022.951} C_VEL
LIN {X 0,Y 594.35,Z 510.452,A -85,B 0,C 180,E1 -1025.41,E2 -1025.41} C_VEL
LIN {X 0,Y 594.389,Z 510.44,A -85,B 0,C 180,E1 -1027.941,E2 -1027.941} C_VEL
LIN {X 0,Y 594.379,Z 510.443,A -85,B 0,C 180,E1 -1030.823,E2 -1030.823} C_VEL
LIN {X 0,Y 594.385,Z 510.442,A -85,B 0,C 180,E1 -1033.842,E2 -1033.842} C_VEL
LIN {X 0,Y 594.368,Z 510.442,A -85,B 0,C 180,E1 -1036.701,E2 -1036.701} C_VEL
LIN {X 0,Y 594.371,Z 510.452,A -85,B 0,C 180,E1 -1039.434,E2 -1039.434} C_VEL
LIN {X 0,Y 594.39,Z 510.439,A -85,B 0,C 180,E1 -1042.392,E2 -1042.392} C_VEL
LIN {X 0,Y 594.398,Z 510.448,A -85,B 0,C 180,E1 -1045.422,E2 -1045.422} C_VEL
LIN {X 0,Y 594.38,Z 510.44,A -85,B 0,C 180,E1 -1048.358,E2 -1048.358} C_VEL
LIN {X 0,Y 594.388,Z 510.442,A -85,B 0,C 180,E1 -1051.043,E2 -1051.043} C_VEL
LIN {X 0,Y 594.381,Z 510.443,A -85,B 0,C 180,E1 -1054.057,E2 -1054.057} C_VEL
LIN {X 0,Y 594.38,Z 510.441,A -85,B 0,C 180,E1 -1056.296,E2 -1056.296} C_VEL
LIN {X 0,Y 594.406,Z 510.441,A -85,B 0,C 180,E1 -1059.225,E2 -1059.225} C_VEL
LIN {X 0,Y 594.355,Z 510.446,A -85,B 0,C 180,E1 -1062.095,E2 -1062.095} C_VEL
LIN {X 0,Y 594.368,Z 510.444,A -85,B 0,C 180,E1 -1064.22,E2 -1064.22} C_VEL
LIN {X 0,Y 594.383,Z 510.441,A -85,B 0,C 180,E1 -1066.321,E2 -1066.321} C_VEL
LIN {X 0,Y 594.378,Z 510.442,A -85,B 0,C 180,E1 -1069.095,E2 -1069.095} C_VEL
LIN {X 0,Y 594.418,Z 510.444,A -85,B 0,C 180,E1 -1071.844,E2 -1071.844} C_VEL
LIN {X 0,Y 594.391,Z 510.439,A -85,B 0,C 180,E1 -1074.573,E2 -1074.573} C_VEL
LIN {X 0,Y 594.413,Z 510.438,A -85,B 0,C 180,E1 -1077.29,E2 -1077.29} C_VEL
LIN {X 0,Y 594.42,Z 510.443,A -85,B 0,C 180,E1 -1080,E2 -1080} C_VEL
LIN {X 0,Y 594.413,Z 510.436,A -85,B 0,C 180,E1 -1082.711,E2 -1082.711} C_VEL
LIN {X 0,Y 594.394,Z 510.442,A -85,B 0,C 180,E1 -1085.428,E2 -1085.428} C_VEL
LIN {X 0,Y 594.418,Z 510.442,A -85,B 0,C 180,E1 -1088.157,E2 -1088.157} C_VEL
LIN {X 0,Y 594.394,Z 510.438,A -85,B 0,C 180,E1 -1091.073,E2 -1091.073} C_VEL
LIN {X 0,Y 594.384,Z 510.445,A -85,B 0,C 180,E1 -1093.679,E2 -1093.679} C_VEL
LIN {X 0,Y 594.399,Z 510.438,A -85,B 0,C 180,E1 -1096.719,E2 -1096.719} C_VEL
LIN {X 0,Y 594.372,Z 510.442,A -85,B 0,C 180,E1 -1099.335,E2 -1099.335} C_VEL
LIN {X 0,Y 594.372,Z 510.443,A -85,B 0,C 180,E1 -1101.503,E2 -1101.503} C_VEL
LIN {X 0,Y 594.397,Z 510.442,A -85,B 0,C 180,E1 -1104.446,E2 -1104.446} C_VEL
LIN {X 0,Y 594.385,Z 510.441,A -85,B 0,C 180,E1 -1106.7,E2 -1106.7} C_VEL
LIN {X 0,Y 594.388,Z 510.439,A -85,B 0,C 180,E1 -1108.998,E2 -1108.998} C_VEL
LIN {X 0,Y 594.383,Z 510.442,A -85,B 0,C 180,E1 -1111.642,E2 -1111.642} C_VEL
LIN {X 0,Y 594.396,Z 510.442,A -85,B 0,C 180,E1 -1114.579,E2 -1114.579} C_VEL
LIN {X 0,Y 594.394,Z 510.44,A -85,B 0,C 180,E1 -1117.608,E2 -1117.608} C_VEL
LIN {X 0,Y 594.371,Z 510.446,A -85,B 0,C 180,E1 -1120.567,E2 -1120.567} C_VEL
LIN {X 0,Y 594.359,Z 510.442,A -85,B 0,C 180,E1 -1123.301,E2 -1123.301} C_VEL
LIN {X 0,Y 594.383,Z 510.448,A -85,B 0,C 180,E1 -1126.159,E2 -1126.159} C_VEL
LIN {X 0,Y 594.381,Z 510.44,A -85,B 0,C 180,E1 -1129.178,E2 -1129.178} C_VEL
LIN {X 0,Y 594.39,Z 510.444,A -85,B 0,C 180,E1 -1132.059,E2 -1132.059} C_VEL
LIN {X 0,Y 594.358,Z 510.448,A -85,B 0,C 180,E1 -1134.676,E2 -1134.676} C_VEL
LIN {X 0,Y 594.384,Z 510.44,A -85,B 0,C 180,E1 -1137.088,E2 -1137.088} C_VEL
LIN {X 0,Y 594.392,Z 510.439,A -85,B 0,C 180,E1 -1139.672,E2 -1139.672} C_VEL
LIN {X 0,Y 594.382,Z 510.45,A -85,B 0,C 180,E1 -1142.539,E2 -1142.539} C_VEL
LIN {X 0,Y 594.379,Z 510.446,A -85,B 0,C 180,E1 -1144.806,E2 -1144.806} C_VEL
LIN {X 0,Y 594.397,Z 510.52,A -85,B 0,C 180,E1 -1147.41,E2 -1147.41} C_VEL
LIN {X 0,Y 594.724,Z 515.496,A -85,B 0,C 180,E1 -1148.145,E2 -1148.145} C_VEL
LIN {X 0,Y 594.594,Z 535.517,A -85,B 0,C 180,E1 -1151.013,E2 -1151.013} C_VEL
LIN {X 0,Y 594.505,Z 554.535,A -85,B 0,C 180,E1 -1153.693,E2 -1153.693} C_VEL
LIN {X 0,Y 594.433,Z 574.684,A -85,B 0,C 180,E1 -1156.496,E2 -1156.496} C_VEL
LIN {X 0,Y 594.47,Z 576.069,A -85,B 0,C 180,E1 -1156.671,E2 -1156.671} C_VEL
LIN {X 0,Y 594.754,Z 583.224,A -85,B 0,C 180,E1 -1156.764,E2 -1156.764} C_VEL
LIN {X 0,Y 594.655,Z 683.899,A -85,B 0,C 180,E1 -1157.998,E2 -1157.998} C_VEL
LIN {X 0,Y 594.616,Z 697.186,A -85,B 0,C 180,E1 -1158.3,E2 -1158.3} C_VEL
LIN {X 0,Y 594.58,Z 709.528,A -85,B 0,C 180,E1 -1158.717,E2 -1158.717} C_VEL
LIN {X 0,Y 594.538,Z 721.616,A -85,B 0,C 180,E1 -1159.269,E2 -1159.269} C_VEL
LIN {X 0,Y 594.468,Z 733.186,A -85,B 0,C 180,E1 -1159.957,E2 -1159.957} C_VEL
LIN {X 0,Y 594.413,Z 743.585,A -85,B 0,C 180,E1 -1160.729,E2 -1160.729} C_VEL
LIN {X 0,Y 594.366,Z 752.103,A -85,B 0,C 180,E1 -1161.499,E2 -1161.499} C_VEL
LIN {X 0,Y 594.348,Z 759.953,A -85,B 0,C 180,E1 -1162.354,E2 -1162.354} C_VEL
LIN {X 0,Y 594.283,Z 767.809,A -85,B 0,C 180,E1 -1163.408,E2 -1163.408} C_VEL
LIN {X 0,Y 594.289,Z 774.675,A -85,B 0,C 180,E1 -1164.57,E2 -1164.57} C_VEL
LIN {X 0,Y 594.27,Z 779.367,A -85,B 0,C 180,E1 -1165.59,E2 -1165.59} C_VEL
LIN {X 0,Y 594.268,Z 782.953,A -85,B 0,C 180,E1 -1166.609,E2 -1166.609} C_VEL
LIN {X 0,Y 594.226,Z 784.806,A -85,B 0,C 180,E1 -1167.287,E2 -1167.287} C_VEL
LIN {X 0,Y 594.239,Z 786.2,A -85,B 0,C 180,E1 -1167.966,E2 -1167.966} C_VEL
LIN {X 0,Y 594.239,Z 787.783,A -85,B 0,C 180,E1 -1169.321,E2 -1169.321} C_VEL
LIN {X 0,Y 594.236,Z 788,A -85,B 0,C 180,E1 -1169.999,E2 -1169.999} C_VEL
LIN {X 0,Y 594.247,Z 787.186,A -85,B 0,C 180,E1 -1171.354,E2 -1171.354} C_VEL
LIN {X 0,Y 594.239,Z 786.203,A -85,B 0,C 180,E1 -1172.032,E2 -1172.032} C_VEL
LIN {X 0,Y 594.226,Z 784.812,A -85,B 0,C 180,E1 -1172.711,E2 -1172.711} C_VEL
LIN {X 0,Y 594.288,Z 781.899,A -85,B 0,C 180,E1 -1173.728,E2 -1173.728} C_VEL
LIN {X 0,Y 594.242,Z 777.954,A -85,B 0,C 180,E1 -1174.748,E2 -1174.748} C_VEL
LIN {X 0,Y 594.304,Z 771.883,A -85,B 0,C 180,E1 -1175.938,E2 -1175.938} C_VEL
LIN {X 0,Y 594.311,Z 765.243,A -85,B 0,C 180,E1 -1176.961,E2 -1176.961} C_VEL
LIN {X 0,Y 594.359,Z 756.999,A -85,B 0,C 180,E1 -1177.985,E2 -1177.985} C_VEL
LIN {X 0,Y 594.382,Z 748.549,A -85,B 0,C 180,E1 -1178.841,E2 -1178.841} C_VEL
LIN {X 0,Y 594.423,Z 738.108,A -85,B 0,C 180,E1 -1179.698,E2 -1179.698} C_VEL
LIN {X 0,Y 594.485,Z 727.776,A -85,B 0,C 180,E1 -1180.385,E2 -1180.385} C_VEL
LIN {X 0,Y 594.56,Z 716.706,A -85,B 0,C 180,E1 -1180.974,E2 -1180.974} C_VEL
LIN {X 0,Y 594.593,Z 704.731,A -85,B 0,C 180,E1 -1181.463,E2 -1181.463} C_VEL
LIN {X 0,Y 594.634,Z 691.397,A -85,B 0,C 180,E1 -1181.849,E2 -1181.849} C_VEL
LIN {X 0,Y 594.69,Z 678.165,A -85,B 0,C 180,E1 -1182.086,E2 -1182.086} C_VEL
LIN {X 0,Y 594.631,Z 577.351,A -85,B 0,C 180,E1 -1183.31,E2 -1183.31} C_VEL
LIN {X 0,Y 594.45,Z 575.8,A -85,B 0,C 180,E1 -1183.35,E2 -1183.35} C_VEL
LIN {X 0,Y 594.505,Z 554.549,A -85,B 0,C 180,E1 -1186.305,E2 -1186.305} C_VEL
LIN {X 0,Y 594.63,Z 534.73,A -85,B 0,C 180,E1 -1189.098,E2 -1189.098} C_VEL
LIN {X 0,Y 594.741,Z 514.251,A -85,B 0,C 180,E1 -1192.035,E2 -1192.035} C_VEL
LIN {X 0,Y 594.388,Z 510.445,A -85,B 0,C 180,E1 -1192.623,E2 -1192.623} C_VEL
LIN {X 0,Y 594.375,Z 510.448,A -85,B 0,C 180,E1 -1195.192,E2 -1195.192} C_VEL
LIN {X 0,Y 594.384,Z 510.451,A -85,B 0,C 180,E1 -1197.526,E2 -1197.526} C_VEL
LIN {X 0,Y 594.386,Z 510.44,A -85,B 0,C 180,E1 -1200.327,E2 -1200.327} C_VEL
LIN {X 0,Y 594.376,Z 510.443,A -85,B 0,C 180,E1 -1202.949,E2 -1202.949} C_VEL
LIN {X 0,Y 594.351,Z 510.454,A -85,B 0,C 180,E1 -1205.407,E2 -1205.407} C_VEL
LIN {X 0,Y 594.386,Z 510.443,A -85,B 0,C 180,E1 -1207.939,E2 -1207.939} C_VEL
LIN {X 0,Y 594.378,Z 510.442,A -85,B 0,C 180,E1 -1210.822,E2 -1210.822} C_VEL
LIN {X 0,Y 594.377,Z 510.445,A -85,B 0,C 180,E1 -1213.84,E2 -1213.84} C_VEL
LIN {X 0,Y 594.36,Z 510.444,A -85,B 0,C 180,E1 -1216.699,E2 -1216.699} C_VEL
LIN {X 0,Y 594.367,Z 510.453,A -85,B 0,C 180,E1 -1219.433,E2 -1219.433} C_VEL
LIN {X 0,Y 594.382,Z 510.44,A -85,B 0,C 180,E1 -1222.39,E2 -1222.39} C_VEL
LIN {X 0,Y 594.381,Z 510.441,A -85,B 0,C 180,E1 -1224.67,E2 -1224.67} C_VEL
LIN {X 0,Y 594.372,Z 510.446,A -85,B 0,C 180,E1 -1227.087,E2 -1227.087} C_VEL
LIN {X 0,Y 594.392,Z 510.445,A -85,B 0,C 180,E1 -1229.668,E2 -1229.668} C_VEL
LIN {X 0,Y 594.364,Z 510.442,A -85,B 0,C 180,E1 -1232.538,E2 -1232.538} C_VEL
LIN {X 0,Y 594.373,Z 510.443,A -85,B 0,C 180,E1 -1234.806,E2 -1234.806} C_VEL
LIN {X 0,Y 594.356,Z 510.45,A -85,B 0,C 180,E1 -1237.263,E2 -1237.263} C_VEL
LIN {X 0,Y 594.37,Z 510.444,A -85,B 0,C 180,E1 -1239.946,E2 -1239.946} C_VEL
LIN {X 0,Y 594.383,Z 510.441,A -85,B 0,C 180,E1 -1242.806,E2 -1242.806} C_VEL
LIN {X 0,Y 594.378,Z 510.445,A -85,B 0,C 180,E1 -1245.825,E2 -1245.825} C_VEL
LIN {X 0,Y 594.385,Z 510.439,A -85,B 0,C 180,E1 -1248.404,E2 -1248.404} C_VEL
LIN {X 0,Y 594.394,Z 510.445,A -85,B 0,C 180,E1 -1251.158,E2 -1251.158} C_VEL
LIN {X 0,Y 594.362,Z 510.446,A -85,B 0,C 180,E1 -1253.891,E2 -1253.891} C_VEL
LIN {X 0,Y 594.378,Z 510.441,A -85,B 0,C 180,E1 -1256.61,E2 -1256.61} C_VEL
LIN {X 0,Y 594.416,Z 510.445,A -85,B 0,C 180,E1 -1259.322,E2 -1259.322} C_VEL
LIN {X 0,Y 594.388,Z 510.441,A -85,B 0,C 180,E1 -1262.032,E2 -1262.032} C_VEL
LIN {X 0,Y 594.396,Z 510.439,A -85,B 0,C 180,E1 -1264.747,E2 -1264.747} C_VEL
LIN {X 0,Y 594.409,Z 510.446,A -85,B 0,C 180,E1 -1267.473,E2 -1267.473} C_VEL
LIN {X 0,Y 594.387,Z 510.44,A -85,B 0,C 180,E1 -1270.216,E2 -1270.216} C_VEL
LIN {X 0,Y 594.365,Z 510.446,A -85,B 0,C 180,E1 -1272.983,E2 -1272.983} C_VEL
LIN {X 0,Y 594.356,Z 510.447,A -85,B 0,C 180,E1 -1275.339,E2 -1275.339} C_VEL
LIN {X 0,Y 593.687,Z 510.531,A -85,B 0,C 180,E1 -1275.905,E2 -1275.905} C_VEL
LIN {X 0,Y 590.832,Z 510.885,A -85,B 0,C 180,E1 -1276.823,E2 -1276.823} C_VEL
LIN {X 0,Y 588.426,Z 511.19,A -85,B 0,C 180,E1 -1277.562,E2 -1277.562} C_VEL
LIN {X 0,Y 587.399,Z 511.312,A -85,B 0,C 180,E1 -1278.132,E2 -1278.132} C_VEL
LIN {X 0,Y 587.318,Z 511.32,A -85,B 0,C 180,E1 -1278.325,E2 -1278.325} C_VEL
LIN {X 0,Y 587.346,Z 511.322,A -85,B 0,C 180,E1 -1281.045,E2 -1281.045} C_VEL
LIN {X 0,Y 587.328,Z 511.321,A -85,B 0,C 180,E1 -1284.006,E2 -1284.006} C_VEL
LIN {X 0,Y 587.354,Z 511.316,A -85,B 0,C 180,E1 -1286.277,E2 -1286.277} C_VEL
LIN {X 0,Y 587.345,Z 511.324,A -85,B 0,C 180,E1 -1289.135,E2 -1289.135} C_VEL
LIN {X 0,Y 587.381,Z 511.374,A -85,B 0,C 180,E1 -1290.455,E2 -1290.455} C_VEL
LIN {X 0,Y 587.503,Z 519.503,A -85,B 0,C 180,E1 -1291.863,E2 -1291.863} C_VEL
LIN {X 0,Y 587.41,Z 535.96,A -85,B 0,C 180,E1 -1294.67,E2 -1294.67} C_VEL
LIN {X 0,Y 587.334,Z 547.184,A -85,B 0,C 180,E1 -1296.562,E2 -1296.562} C_VEL
LIN {X 0,Y 587.855,Z 551.963,A -85,B 0,C 180,E1 -1296.635,E2 -1296.635} C_VEL
LIN {X 0,Y 587.744,Z 654.113,A -85,B 0,C 180,E1 -1297.903,E2 -1297.903} C_VEL
LIN {X 0,Y 587.683,Z 667.436,A -85,B 0,C 180,E1 -1298.212,E2 -1298.212} C_VEL
LIN {X 0,Y 587.617,Z 679.957,A -85,B 0,C 180,E1 -1298.643,E2 -1298.643} C_VEL
LIN {X 0,Y 587.552,Z 691.46,A -85,B 0,C 180,E1 -1299.177,E2 -1299.177} C_VEL
LIN {X 0,Y 587.437,Z 703.253,A -85,B 0,C 180,E1 -1299.884,E2 -1299.884} C_VEL
LIN {X 0,Y 587.379,Z 714.049,A -85,B 0,C 180,E1 -1300.699,E2 -1300.699} C_VEL
LIN {X 0,Y 587.325,Z 723.781,A -85,B 0,C 180,E1 -1301.614,E2 -1301.614} C_VEL
LIN {X 0,Y 587.248,Z 731.843,A -85,B 0,C 180,E1 -1302.544,E2 -1302.544} C_VEL
LIN {X 0,Y 587.223,Z 738.693,A -85,B 0,C 180,E1 -1303.508,E2 -1303.508} C_VEL
LIN {X 0,Y 587.224,Z 745.456,A -85,B 0,C 180,E1 -1304.702,E2 -1304.702} C_VEL
LIN {X 0,Y 587.174,Z 750.591,A -85,B 0,C 180,E1 -1305.901,E2 -1305.901} C_VEL
LIN {X 0,Y 587.163,Z 753.992,A -85,B 0,C 180,E1 -1306.982,E2 -1306.982} C_VEL
LIN {X 0,Y 587.152,Z 756.08,A -85,B 0,C 180,E1 -1307.912,E2 -1307.912} C_VEL
LIN {X 0,Y 587.115,Z 757.494,A -85,B 0,C 180,E1 -1308.949,E2 -1308.949} C_VEL
LIN {X 0,Y 587.135,Z 757.996,A -85,B 0,C 180,E1 -1310.002,E2 -1310.002} C_VEL
LIN {X 0,Y 587.108,Z 757.543,A -85,B 0,C 180,E1 -1311.085,E2 -1311.085} C_VEL
LIN {X 0,Y 587.136,Z 755.683,A -85,B 0,C 180,E1 -1312.378,E2 -1312.378} C_VEL
LIN {X 0,Y 587.182,Z 752.244,A -85,B 0,C 180,E1 -1313.709,E2 -1313.709} C_VEL
LIN {X 0,Y 587.164,Z 747.58,A -85,B 0,C 180,E1 -1314.935,E2 -1314.935} C_VEL
LIN {X 0,Y 587.22,Z 741.125,A -85,B 0,C 180,E1 -1316.186,E2 -1316.186} C_VEL
LIN {X 0,Y 587.243,Z 734.766,A -85,B 0,C 180,E1 -1317.158,E2 -1317.158} C_VEL
LIN {X 0,Y 587.3,Z 726.083,A -85,B 0,C 180,E1 -1318.23,E2 -1318.23} C_VEL
LIN {X 0,Y 587.365,Z 716.649,A -85,B 0,C 180,E1 -1319.164,E2 -1319.164} C_VEL
LIN {X 0,Y 587.436,Z 705.739,A -85,B 0,C 180,E1 -1320.035,E2 -1320.035} C_VEL
LIN {X 0,Y 587.499,Z 694.104,A -85,B 0,C 180,E1 -1320.768,E2 -1320.768} C_VEL
LIN {X 0,Y 587.595,Z 681.713,A -85,B 0,C 180,E1 -1321.375,E2 -1321.375} C_VEL
LIN {X 0,Y 587.651,Z 668.938,A -85,B 0,C 180,E1 -1321.835,E2 -1321.835} C_VEL
LIN {X 0,Y 587.734,Z 655.777,A -85,B 0,C 180,E1 -1322.155,E2 -1322.155} C_VEL
LIN {X 0,Y 587.758,Z 629.328,A -85,B 0,C 180,E1 -1322.507,E2 -1322.507} C_VEL
LIN {X 0,Y 587.693,Z 549.475,A -85,B 0,C 180,E1 -1323.489,E2 -1323.489} C_VEL
LIN {X 0,Y 587.347,Z 547.039,A -85,B 0,C 180,E1 -1323.552,E2 -1323.552} C_VEL
LIN {X 0,Y 587.428,Z 531.446,A -85,B 0,C 180,E1 -1326.186,E2 -1326.186} C_VEL
LIN {X 0,Y 587.541,Z 514.115,A -85,B 0,C 180,E1 -1329.155,E2 -1329.155} C_VEL
LIN {X 0,Y 587.33,Z 511.323,A -85,B 0,C 180,E1 -1329.651,E2 -1329.651} C_VEL
LIN {X 0,Y 587.355,Z 511.324,A -85,B 0,C 180,E1 -1332.595,E2 -1332.595} C_VEL
LIN {X 0,Y 587.361,Z 511.315,A -85,B 0,C 180,E1 -1335.74,E2 -1335.74} C_VEL
LIN {X 0,Y 587.343,Z 511.327,A -85,B 0,C 180,E1 -1338.867,E2 -1338.867} C_VEL
LIN {X 0,Y 587.363,Z 511.314,A -85,B 0,C 180,E1 -1341.746,E2 -1341.746} C_VEL
LIN {X 0,Y 587.364,Z 511.319,A -85,B 0,C 180,E1 -1344.508,E2 -1344.508} C_VEL
LIN {X 0,Y 587.369,Z 511.318,A -85,B 0,C 180,E1 -1347.258,E2 -1347.258} C_VEL
LIN {X 0,Y 587.383,Z 511.312,A -85,B 0,C 180,E1 -1350.001,E2 -1350.001} C_VEL
LIN {X 0,Y 587.371,Z 511.32,A -85,B 0,C 180,E1 -1352.744,E2 -1352.744} C_VEL
LIN {X 0,Y 587.359,Z 511.317,A -85,B 0,C 180,E1 -1355.494,E2 -1355.494} C_VEL
LIN {X 0,Y 587.364,Z 511.315,A -85,B 0,C 180,E1 -1358.256,E2 -1358.256} C_VEL
LIN {X 0,Y 587.347,Z 511.325,A -85,B 0,C 180,E1 -1361.135,E2 -1361.135} C_VEL
LIN {X 0,Y 587.364,Z 511.314,A -85,B 0,C 180,E1 -1364.261,E2 -1364.261} C_VEL
LIN {X 0,Y 587.346,Z 511.321,A -85,B 0,C 180,E1 -1367.407,E2 -1367.407} C_VEL
LIN {X 0,Y 587.327,Z 511.319,A -85,B 0,C 180,E1 -1370.306,E2 -1370.306} C_VEL
LIN {X 0,Y 587.315,Z 511.329,A -85,B 0,C 180,E1 -1373.26,E2 -1373.26} C_VEL
LIN {X 0,Y 587.332,Z 511.323,A -85,B 0,C 180,E1 -1375.518,E2 -1375.518} C_VEL
LIN {X 0,Y 587.347,Z 511.318,A -85,B 0,C 180,E1 -1377.819,E2 -1377.819} C_VEL
LIN {X 0,Y 587.344,Z 511.317,A -85,B 0,C 180,E1 -1380.512,E2 -1380.512} C_VEL
LIN {X 0,Y 587.34,Z 511.325,A -85,B 0,C 180,E1 -1383.113,E2 -1383.113} C_VEL
LIN {X 0,Y 587.298,Z 511.328,A -85,B 0,C 180,E1 -1385.538,E2 -1385.538} C_VEL
LIN {X 0,Y 587.343,Z 511.319,A -85,B 0,C 180,E1 -1387.84,E2 -1387.84} C_VEL
LIN {X 0,Y 587.319,Z 511.319,A -85,B 0,C 180,E1 -1390.255,E2 -1390.255} C_VEL
LIN {X 0,Y 587.324,Z 511.324,A -85,B 0,C 180,E1 -1393.006,E2 -1393.006} C_VEL
LIN {X 0,Y 587.329,Z 511.321,A -85,B 0,C 180,E1 -1395.887,E2 -1395.887} C_VEL
LIN {X 0,Y 587.337,Z 511.32,A -85,B 0,C 180,E1 -1398.926,E2 -1398.926} C_VEL
LIN {X 0,Y 587.333,Z 511.327,A -85,B 0,C 180,E1 -1401.521,E2 -1401.521} C_VEL
LIN {X 0,Y 587.296,Z 511.324,A -85,B 0,C 180,E1 -1404.101,E2 -1404.101} C_VEL
LIN {X 0,Y 587.338,Z 511.317,A -85,B 0,C 180,E1 -1406.604,E2 -1406.604} C_VEL
LIN {X 0,Y 587.339,Z 511.328,A -85,B 0,C 180,E1 -1409.491,E2 -1409.491} C_VEL
LIN {X 0,Y 587.346,Z 511.317,A -85,B 0,C 180,E1 -1412.309,E2 -1412.309} C_VEL
LIN {X 0,Y 587.34,Z 511.317,A -85,B 0,C 180,E1 -1414.484,E2 -1414.484} C_VEL
LIN {X 0,Y 587.343,Z 511.325,A -85,B 0,C 180,E1 -1417.487,E2 -1417.487} C_VEL
LIN {X 0,Y 587.317,Z 511.32,A -85,B 0,C 180,E1 -1420.424,E2 -1420.424} C_VEL
LIN {X 0,Y 587.358,Z 511.319,A -85,B 0,C 180,E1 -1423.312,E2 -1423.312} C_VEL
LIN {X 0,Y 587.362,Z 511.317,A -85,B 0,C 180,E1 -1426.155,E2 -1426.155} C_VEL
LIN {X 0,Y 587.344,Z 511.317,A -85,B 0,C 180,E1 -1428.963,E2 -1428.963} C_VEL
LIN {X 0,Y 587.37,Z 511.324,A -85,B 0,C 180,E1 -1431.745,E2 -1431.745} C_VEL
LIN {X 0,Y 587.357,Z 511.315,A -85,B 0,C 180,E1 -1434.507,E2 -1434.507} C_VEL
LIN {X 0,Y 587.379,Z 511.314,A -85,B 0,C 180,E1 -1437.257,E2 -1437.257} C_VEL
LIN {X 0,Y 587.389,Z 511.318,A -85,B 0,C 180,E1 -1440,E2 -1440} C_VEL
LIN {X 0,Y 587.379,Z 511.312,A -85,B 0,C 180,E1 -1442.744,E2 -1442.744} C_VEL
LIN {X 0,Y 587.36,Z 511.319,A -85,B 0,C 180,E1 -1445.493,E2 -1445.493} C_VEL
LIN {X 0,Y 587.37,Z 511.318,A -85,B 0,C 180,E1 -1448.256,E2 -1448.256} C_VEL
LIN {X 0,Y 587.356,Z 511.315,A -85,B 0,C 180,E1 -1451.134,E2 -1451.134} C_VEL
LIN {X 0,Y 587.372,Z 511.319,A -85,B 0,C 180,E1 -1454.26,E2 -1454.26} C_VEL
LIN {X 0,Y 587.354,Z 511.317,A -85,B 0,C 180,E1 -1457.406,E2 -1457.406} C_VEL
LIN {X 0,Y 587.334,Z 511.324,A -85,B 0,C 180,E1 -1460.305,E2 -1460.305} C_VEL
LIN {X 0,Y 587.322,Z 511.32,A -85,B 0,C 180,E1 -1463.259,E2 -1463.259} C_VEL
LIN {X 0,Y 587.339,Z 511.319,A -85,B 0,C 180,E1 -1465.517,E2 -1465.517} C_VEL
LIN {X 0,Y 587.347,Z 511.322,A -85,B 0,C 180,E1 -1467.818,E2 -1467.818} C_VEL
LIN {X 0,Y 587.343,Z 511.321,A -85,B 0,C 180,E1 -1470.51,E2 -1470.51} C_VEL
LIN {X 0,Y 587.334,Z 511.318,A -85,B 0,C 180,E1 -1473.397,E2 -1473.397} C_VEL
LIN {X 0,Y 587.307,Z 511.327,A -85,B 0,C 180,E1 -1475.899,E2 -1475.899} C_VEL
LIN {X 0,Y 587.335,Z 511.324,A -85,B 0,C 180,E1 -1478.479,E2 -1478.479} C_VEL
LIN {X 0,Y 587.34,Z 511.317,A -85,B 0,C 180,E1 -1481.157,E2 -1481.157} C_VEL
LIN {X 0,Y 587.31,Z 511.329,A -85,B 0,C 180,E1 -1484.111,E2 -1484.111} C_VEL
LIN {X 0,Y 587.327,Z 511.319,A -85,B 0,C 180,E1 -1486.994,E2 -1486.994} C_VEL
LIN {X 0,Y 587.318,Z 511.322,A -85,B 0,C 180,E1 -1489.745,E2 -1489.745} C_VEL
LIN {X 0,Y 587.351,Z 511.326,A -85,B 0,C 180,E1 -1492.392,E2 -1492.392} C_VEL
LIN {X 0,Y 587.365,Z 511.315,A -85,B 0,C 180,E1 -1495.779,E2 -1495.779} C_VEL
LIN {X 0,Y 587.347,Z 511.324,A -85,B 0,C 180,E1 -1498.231,E2 -1498.231} C_VEL
LIN {X 0,Y 587.355,Z 511.319,A -85,B 0,C 180,E1 -1500.866,E2 -1500.866} C_VEL
LIN {X 0,Y 587.342,Z 511.318,A -85,B 0,C 180,E1 -1503.721,E2 -1503.721} C_VEL
LIN {X 0,Y 587.341,Z 511.321,A -85,B 0,C 180,E1 -1505.993,E2 -1505.993} C_VEL
LIN {X 0,Y 587.348,Z 511.439,A -85,B 0,C 180,E1 -1507.259,E2 -1507.259} C_VEL
LIN {X 0,Y 587.824,Z 515.496,A -85,B 0,C 180,E1 -1507.875,E2 -1507.875} C_VEL
LIN {X 0,Y 587.673,Z 536.128,A -85,B 0,C 180,E1 -1510.868,E2 -1510.868} C_VEL
LIN {X 0,Y 587.512,Z 555.794,A -85,B 0,C 180,E1 -1513.672,E2 -1513.672} C_VEL
LIN {X 0,Y 587.389,Z 575.786,A -85,B 0,C 180,E1 -1516.485,E2 -1516.485} C_VEL
LIN {X 0,Y 587.887,Z 579.647,A -85,B 0,C 180,E1 -1516.563,E2 -1516.563} C_VEL
LIN {X 0,Y 587.733,Z 683.899,A -85,B 0,C 180,E1 -1517.854,E2 -1517.854} C_VEL
LIN {X 0,Y 587.667,Z 697.187,A -85,B 0,C 180,E1 -1518.159,E2 -1518.159} C_VEL
LIN {X 0,Y 587.627,Z 709.734,A -85,B 0,C 180,E1 -1518.589,E2 -1518.589} C_VEL
LIN {X 0,Y 587.54,Z 721.615,A -85,B 0,C 180,E1 -1519.14,E2 -1519.14} C_VEL
LIN {X 0,Y 587.458,Z 733.187,A -85,B 0,C 180,E1 -1519.835,E2 -1519.835} C_VEL
LIN {X 0,Y 587.391,Z 743.586,A -85,B 0,C 180,E1 -1520.617,E2 -1520.617} C_VEL
LIN {X 0,Y 587.31,Z 752.103,A -85,B 0,C 180,E1 -1521.396,E2 -1521.396} C_VEL
LIN {X 0,Y 587.274,Z 759.953,A -85,B 0,C 180,E1 -1522.262,E2 -1522.262} C_VEL
LIN {X 0,Y 587.231,Z 766.463,A -85,B 0,C 180,E1 -1523.125,E2 -1523.125} C_VEL
LIN {X 0,Y 587.236,Z 772.861,A -85,B 0,C 180,E1 -1524.16,E2 -1524.16} C_VEL
LIN {X 0,Y 587.147,Z 777.946,A -85,B 0,C 180,E1 -1525.193,E2 -1525.193} C_VEL
LIN {X 0,Y 587.212,Z 781.893,A -85,B 0,C 180,E1 -1526.225,E2 -1526.225} C_VEL
LIN {X 0,Y 587.132,Z 784.806,A -85,B 0,C 180,E1 -1527.255,E2 -1527.255} C_VEL
LIN {X 0,Y 587.138,Z 786.199,A -85,B 0,C 180,E1 -1527.941,E2 -1527.941} C_VEL
LIN {X 0,Y 587.14,Z 787.784,A -85,B 0,C 180,E1 -1529.313,E2 -1529.313} C_VEL
LIN {X 0,Y 587.137,Z 788,A -85,B 0,C 180,E1 -1529.999,E2 -1529.999} C_VEL
LIN {X 0,Y 587.147,Z 787.186,A -85,B 0,C 180,E1 -1531.371,E2 -1531.371} C_VEL
LIN {X 0,Y 587.138,Z 786.203,A -85,B 0,C 180,E1 -1532.057,E2 -1532.057} C_VEL
LIN {X 0,Y 587.132,Z 784.812,A -85,B 0,C 180,E1 -1532.743,E2 -1532.743} C_VEL
LIN {X 0,Y 587.212,Z 781.899,A -85,B 0,C 180,E1 -1533.773,E2 -1533.773} C_VEL
LIN {X 0,Y 587.147,Z 777.954,A -85,B 0,C 180,E1 -1534.805,E2 -1534.805} C_VEL
LIN {X 0,Y 587.217,Z 771.883,A -85,B 0,C 180,E1 -1536.01,E2 -1536.01} C_VEL
LIN {X 0,Y 587.246,Z 765.244,A -85,B 0,C 180,E1 -1537.045,E2 -1537.045} C_VEL
LIN {X 0,Y 587.299,Z 756.999,A -85,B 0,C 180,E1 -1538.082,E2 -1538.082} C_VEL
LIN {X 0,Y 587.343,Z 748.549,A -85,B 0,C 180,E1 -1538.948,E2 -1538.948} C_VEL
LIN {X 0,Y 587.41,Z 738.109,A -85,B 0,C 180,E1 -1539.815,E2 -1539.815} C_VEL
LIN {X 0,Y 587.504,Z 727.776,A -85,B 0,C 180,E1 -1540.51,E2 -1540.51} C_VEL
LIN {X 0,Y 587.582,Z 715.821,A -85,B 0,C 180,E1 -1541.148,E2 -1541.148} C_VEL
LIN {X 0,Y 587.623,Z 703.621,A -85,B 0,C 180,E1 -1541.639,E2 -1541.639} C_VEL
LIN {X 0,Y 587.708,Z 690.482,A -85,B 0,C 180,E1 -1542.013,E2 -1542.013} C_VEL
LIN {X 0,Y 587.758,Z 678.165,A -85,B 0,C 180,E1 -1542.231,E2 -1542.231} C_VEL
LIN {X 0,Y 587.712,Z 577.919,A -85,B 0,C 180,E1 -1543.463,E2 -1543.463} C_VEL
LIN {X 0,Y 587.389,Z 575.8,A -85,B 0,C 180,E1 -1543.513,E2 -1543.513} C_VEL
LIN {X 0,Y 587.494,Z 557.068,A -85,B 0,C 180,E1 -1546.148,E2 -1546.148} C_VEL
LIN {X 0,Y 587.601,Z 539.437,A -85,B 0,C 180,E1 -1548.658,E2 -1548.658} C_VEL
LIN {X 0,Y 587.79,Z 520.532,A -85,B 0,C 180,E1 -1551.389,E2 -1551.389} C_VEL
LIN {X 0,Y 587.655,Z 512.992,A -85,B 0,C 180,E1 -1552.5,E2 -1552.5} C_VEL
LIN {X 0,Y 587.33,Z 511.326,A -85,B 0,C 180,E1 -1552.791,E2 -1552.791} C_VEL
LIN {X 0,Y 587.332,Z 511.329,A -85,B 0,C 180,E1 -1555.515,E2 -1555.515} C_VEL
LIN {X 0,Y 587.347,Z 511.322,A -85,B 0,C 180,E1 -1557.816,E2 -1557.816} C_VEL
LIN {X 0,Y 587.341,Z 511.318,A -85,B 0,C 180,E1 -1560.51,E2 -1560.51} C_VEL
LIN {X 0,Y 587.338,Z 511.322,A -85,B 0,C 180,E1 -1563.111,E2 -1563.111} C_VEL
LIN {X 0,Y 587.315,Z 511.324,A -85,B 0,C 180,E1 -1565.897,E2 -1565.897} C_VEL
LIN {X 0,Y 587.33,Z 511.319,A -85,B 0,C 180,E1 -1568.478,E2 -1568.478} C_VEL
LIN {X 0,Y 587.335,Z 511.324,A -85,B 0,C 180,E1 -1571.155,E2 -1571.155} C_VEL
LIN {X 0,Y 587.329,Z 511.32,A -85,B 0,C 180,E1 -1574.113,E2 -1574.113} C_VEL
LIN {X 0,Y 587.308,Z 511.325,A -85,B 0,C 180,E1 -1576.993,E2 -1576.993} C_VEL
LIN {X 0,Y 587.315,Z 511.326,A -85,B 0,C 180,E1 -1579.745,E2 -1579.745} C_VEL
LIN {X 0,Y 587.338,Z 511.317,A -85,B 0,C 180,E1 -1582.391,E2 -1582.391} C_VEL
LIN {X 0,Y 587.346,Z 511.319,A -85,B 0,C 180,E1 -1584.945,E2 -1584.945} C_VEL
LIN {X 0,Y 587.334,Z 511.328,A -85,B 0,C 180,E1 -1587.42,E2 -1587.42} C_VEL
LIN {X 0,Y 587.339,Z 511.322,A -85,B 0,C 180,E1 -1589.83,E2 -1589.83} C_VEL
LIN {X 0,Y 587.343,Z 511.317,A -85,B 0,C 180,E1 -1592.306,E2 -1592.306} C_VEL
LIN {X 0,Y 587.334,Z 511.318,A -85,B 0,C 180,E1 -1594.483,E2 -1594.483} C_VEL
LIN {X 0,Y 587.332,Z 511.328,A -85,B 0,C 180,E1 -1597.486,E2 -1597.486} C_VEL
LIN {X 0,Y 587.325,Z 511.324,A -85,B 0,C 180,E1 -1599.695,E2 -1599.695} C_VEL
LIN {X 0,Y 587.35,Z 511.316,A -85,B 0,C 180,E1 -1602.594,E2 -1602.594} C_VEL
LIN {X 0,Y 587.354,Z 511.321,A -85,B 0,C 180,E1 -1605.739,E2 -1605.739} C_VEL
LIN {X 0,Y 587.352,Z 511.317,A -85,B 0,C 180,E1 -1608.858,E2 -1608.858} C_VEL
LIN {X 0,Y 587.363,Z 511.319,A -85,B 0,C 180,E1 -1611.744,E2 -1611.744} C_VEL
LIN {X 0,Y 587.351,Z 511.316,A -85,B 0,C 180,E1 -1614.507,E2 -1614.507} C_VEL
LIN {X 0,Y 587.376,Z 511.321,A -85,B 0,C 180,E1 -1617.256,E2 -1617.256} C_VEL
LIN {X 0,Y 587.373,Z 511.315,A -85,B 0,C 180,E1 -1620,E2 -1620} C_VEL
LIN {X 0,Y 587.374,Z 511.314,A -85,B 0,C 180,E1 -1622.743,E2 -1622.743} C_VEL
LIN {X 0,Y 587.351,Z 511.325,A -85,B 0,C 180,E1 -1625.493,E2 -1625.493} C_VEL
LIN {X 0,Y 587.363,Z 511.315,A -85,B 0,C 180,E1 -1628.255,E2 -1628.255} C_VEL
LIN {X 0,Y 587.35,Z 511.322,A -85,B 0,C 180,E1 -1631.141,E2 -1631.141} C_VEL
LIN {X 0,Y 587.353,Z 511.316,A -85,B 0,C 180,E1 -1634.261,E2 -1634.261} C_VEL
LIN {X 0,Y 587.35,Z 511.327,A -85,B 0,C 180,E1 -1637.406,E2 -1637.406} C_VEL
LIN {X 0,Y 587.318,Z 511.32,A -85,B 0,C 180,E1 -1638.325,E2 -1638.325} C_VEL
LIN {X 0,Y 586.666,Z 511.405,A -85,B 0,C 180,E1 -1638.897,E2 -1638.897} C_VEL
LIN {X 0,Y 583.834,Z 511.766,A -85,B 0,C 180,E1 -1639.825,E2 -1639.825} C_VEL
LIN {X 0,Y 581.424,Z 512.07,A -85,B 0,C 180,E1 -1640.572,E2 -1640.572} C_VEL
LIN {X 0,Y 580.372,Z 512.197,A -85,B 0,C 180,E1 -1641.149,E2 -1641.149} C_VEL
LIN {X 0,Y 580.277,Z 512.206,A -85,B 0,C 180,E1 -1641.344,E2 -1641.344} C_VEL
LIN {X 0,Y 580.29,Z 512.196,A -85,B 0,C 180,E1 -1644.316,E2 -1644.316} C_VEL
LIN {X 0,Y 580.3,Z 512.196,A -85,B 0,C 180,E1 -1646.622,E2 -1646.622} C_VEL
LIN {X 0,Y 580.297,Z 512.205,A -85,B 0,C 180,E1 -1649.312,E2 -1649.312} C_VEL
LIN {X 0,Y 580.337,Z 512.306,A -85,B 0,C 180,E1 -1650.371,E2 -1650.371} C_VEL
LIN {X 0,Y 580.506,Z 519.961,A -85,B 0,C 180,E1 -1651.716,E2 -1651.716} C_VEL
LIN {X 0,Y 580.389,Z 537.182,A -85,B 0,C 180,E1 -1654.689,E2 -1654.689} C_VEL
LIN {X 0,Y 580.307,Z 547.373,A -85,B 0,C 180,E1 -1656.4,E2 -1656.4} C_VEL
LIN {X 0,Y 580.953,Z 551.91,A -85,B 0,C 180,E1 -1656.472,E2 -1656.472} C_VEL
LIN {X 0,Y 580.808,Z 654.438,A -85,B 0,C 180,E1 -1657.762,E2 -1657.762} C_VEL
LIN {X 0,Y 580.729,Z 667.503,A -85,B 0,C 180,E1 -1658.07,E2 -1658.07} C_VEL
LIN {X 0,Y 580.648,Z 680.251,A -85,B 0,C 180,E1 -1658.516,E2 -1658.516} C_VEL
LIN {X 0,Y 580.574,Z 692.099,A -85,B 0,C 180,E1 -1659.08,E2 -1659.08} C_VEL
LIN {X 0,Y 580.439,Z 702.808,A -85,B 0,C 180,E1 -1659.729,E2 -1659.729} C_VEL
LIN {X 0,Y 580.347,Z 713.415,A -85,B 0,C 180,E1 -1660.532,E2 -1660.532} C_VEL
LIN {X 0,Y 580.291,Z 722.089,A -85,B 0,C 180,E1 -1661.334,E2 -1661.334} C_VEL
LIN {X 0,Y 580.187,Z 731.151,A -85,B 0,C 180,E1 -1662.363,E2 -1662.363} C_VEL
LIN {X 0,Y 580.153,Z 738.385,A -85,B 0,C 180,E1 -1663.38,E2 -1663.38} C_VEL
LIN {X 0,Y 580.136,Z 744.148,A -85,B 0,C 180,E1 -1664.379,E2 -1664.379} C_VEL
LIN {X 0,Y 580.103,Z 748.691,A -85,B 0,C 180,E1 -1665.36,E2 -1665.36} C_VEL
LIN {X 0,Y 580.062,Z 753.138,A -85,B 0,C 180,E1 -1666.631,E2 -1666.631} C_VEL
LIN {X 0,Y 580.061,Z 755.62,A -85,B 0,C 180,E1 -1667.652,E2 -1667.652} C_VEL
LIN {X 0,Y 580.028,Z 757.23,A -85,B 0,C 180,E1 -1668.697,E2 -1668.697} C_VEL
LIN {X 0,Y 580.041,Z 758,A -85,B 0,C 180,E1 -1670.048,E2 -1670.048} C_VEL
LIN {X 0,Y 580.007,Z 757.646,A -85,B 0,C 180,E1 -1670.945,E2 -1670.945} C_VEL
LIN {X 0,Y 580.014,Z 756.466,A -85,B 0,C 180,E1 -1671.961,E2 -1671.961} C_VEL
LIN {X 0,Y 580.05,Z 754.115,A -85,B 0,C 180,E1 -1673.098,E2 -1673.098} C_VEL
LIN {X 0,Y 580.101,Z 749.841,A -85,B 0,C 180,E1 -1674.444,E2 -1674.444} C_VEL
LIN {X 0,Y 580.08,Z 745.364,A -85,B 0,C 180,E1 -1675.472,E2 -1675.472} C_VEL
LIN {X 0,Y 580.147,Z 740.036,A -85,B 0,C 180,E1 -1676.447,E2 -1676.447} C_VEL
LIN {X 0,Y 580.191,Z 732.222,A -85,B 0,C 180,E1 -1677.589,E2 -1677.589} C_VEL
LIN {X 0,Y 580.279,Z 723.432,A -85,B 0,C 180,E1 -1678.616,E2 -1678.616} C_VEL
LIN {X 0,Y 580.349,Z 713.75,A -85,B 0,C 180,E1 -1679.53,E2 -1679.53} C_VEL
LIN {X 0,Y 580.456,Z 702.798,A -85,B 0,C 180,E1 -1680.361,E2 -1680.361} C_VEL
LIN {X 0,Y 580.569,Z 691.548,A -85,B 0,C 180,E1 -1681.04,E2 -1681.04} C_VEL
LIN {X 0,Y 580.657,Z 679.888,A -85,B 0,C 180,E1 -1681.589,E2 -1681.589} C_VEL
LIN {X 0,Y 580.716,Z 666.484,A -85,B 0,C 180,E1 -1682.05,E2 -1682.05} C_VEL
LIN {X 0,Y 580.78,Z 654.01,A -85,B 0,C 180,E1 -1682.337,E2 -1682.337} C_VEL
LIN {X 0,Y 580.902,Z 550.956,A -85,B 0,C 180,E1 -1683.631,E2 -1683.631} C_VEL
LIN {X 0,Y 580.313,Z 547.07,A -85,B 0,C 180,E1 -1683.713,E2 -1683.713} C_VEL
LIN {X 0,Y 580.411,Z 531.085,A -85,B 0,C 180,E1 -1686.449,E2 -1686.449} C_VEL
LIN {X 0,Y 580.556,Z 515.741,A -85,B 0,C 180,E1 -1689.109,E2 -1689.109} C_VEL
LIN {X 0,Y 580.288,Z 512.201,A -85,B 0,C 180,E1 -1689.763,E2 -1689.763} C_VEL
LIN {X 0,Y 580.301,Z 512.2,A -85,B 0,C 180,E1 -1692.377,E2 -1692.377} C_VEL
LIN {X 0,Y 580.283,Z 512.199,A -85,B 0,C 180,E1 -1695.267,E2 -1695.267} C_VEL
LIN {X 0,Y 580.307,Z 512.194,A -85,B 0,C 180,E1 -1698.12,E2 -1698.12} C_VEL
LIN {X 0,Y 580.279,Z 512.205,A -85,B 0,C 180,E1 -1700.942,E2 -1700.942} C_VEL
LIN {X 0,Y 580.308,Z 512.197,A -85,B 0,C 180,E1 -1703.254,E2 -1703.254} C_VEL
LIN {X 0,Y 580.272,Z 512.197,A -85,B 0,C 180,E1 -1705.834,E2 -1705.834} C_VEL
LIN {X 0,Y 580.342,Z 512.189,A -85,B 0,C 180,E1 -1707.919,E2 -1707.919} C_VEL
LIN {X 0,Y 580.361,Z 512.193,A -85,B 0,C 180,E1 -1710.695,E2 -1710.695} C_VEL
LIN {X 0,Y 580.282,Z 512.199,A -85,B 0,C 180,E1 -1713.473,E2 -1713.473} C_VEL
LIN {X 0,Y 580.326,Z 512.193,A -85,B 0,C 180,E1 -1715.561,E2 -1715.561} C_VEL
LIN {X 0,Y 580.327,Z 512.192,A -85,B 0,C 180,E1 -1718.357,E2 -1718.357} C_VEL
LIN {X 0,Y 580.299,Z 512.202,A -85,B 0,C 180,E1 -1721.192,E2 -1721.192} C_VEL
LIN {X 0,Y 580.326,Z 512.191,A -85,B 0,C 180,E1 -1724.018,E2 -1724.018} C_VEL
LIN {X 0,Y 580.312,Z 512.2,A -85,B 0,C 180,E1 -1726.915,E2 -1726.915} C_VEL
LIN {X 0,Y 580.304,Z 512.194,A -85,B 0,C 180,E1 -1729.823,E2 -1729.823} C_VEL
LIN {X 0,Y 580.291,Z 512.2,A -85,B 0,C 180,E1 -1732.803,E2 -1732.803} C_VEL
LIN {X 0,Y 580.306,Z 512.202,A -85,B 0,C 180,E1 -1735.081,E2 -1735.081} C_VEL
LIN {X 0,Y 580.299,Z 512.194,A -85,B 0,C 180,E1 -1738.186,E2 -1738.186} C_VEL
LIN {X 0,Y 580.294,Z 512.197,A -85,B 0,C 180,E1 -1740.697,E2 -1740.697} C_VEL
LIN {X 0,Y 580.305,Z 512.203,A -85,B 0,C 180,E1 -1743.317,E2 -1743.317} C_VEL
LIN {X 0,Y 580.247,Z 512.204,A -85,B 0,C 180,E1 -1745.757,E2 -1745.757} C_VEL
LIN {X 0,Y 580.291,Z 512.195,A -85,B 0,C 180,E1 -1748.147,E2 -1748.147} C_VEL
LIN {X 0,Y 580.301,Z 512.197,A -85,B 0,C 180,E1 -1750.844,E2 -1750.844} C_VEL
LIN {X 0,Y 580.29,Z 512.201,A -85,B 0,C 180,E1 -1753.658,E2 -1753.658} C_VEL
LIN {X 0,Y 580.278,Z 512.197,A -85,B 0,C 180,E1 -1756.61,E2 -1756.61} C_VEL
LIN {X 0,Y 580.301,Z 512.2,A -85,B 0,C 180,E1 -1759.157,E2 -1759.157} C_VEL
LIN {X 0,Y 580.292,Z 512.198,A -85,B 0,C 180,E1 -1761.928,E2 -1761.928} C_VEL
LIN {X 0,Y 580.26,Z 512.199,A -85,B 0,C 180,E1 -1764.454,E2 -1764.454} C_VEL
LIN {X 0,Y 580.295,Z 512.197,A -85,B 0,C 180,E1 -1766.976,E2 -1766.976} C_VEL
LIN {X 0,Y 580.298,Z 512.203,A -85,B 0,C 180,E1 -1769.426,E2 -1769.426} C_VEL
LIN {X 0,Y 580.297,Z 512.196,A -85,B 0,C 180,E1 -1772.143,E2 -1772.143} C_VEL
LIN {X 0,Y 580.312,Z 512.194,A -85,B 0,C 180,E1 -1774.921,E2 -1774.921} C_VEL
LIN {X 0,Y 580.276,Z 512.202,A -85,B 0,C 180,E1 -1777.948,E2 -1777.948} C_VEL
LIN {X 0,Y 580.303,Z 512.194,A -85,B 0,C 180,E1 -1780.914,E2 -1780.914} C_VEL
LIN {X 0,Y 580.284,Z 512.204,A -85,B 0,C 180,E1 -1783.826,E2 -1783.826} C_VEL
LIN {X 0,Y 580.33,Z 512.196,A -85,B 0,C 180,E1 -1785.984,E2 -1785.984} C_VEL
LIN {X 0,Y 580.311,Z 512.193,A -85,B 0,C 180,E1 -1788.827,E2 -1788.827} C_VEL
LIN {X 0,Y 580.333,Z 512.199,A -85,B 0,C 180,E1 -1791.644,E2 -1791.644} C_VEL
LIN {X 0,Y 580.324,Z 512.192,A -85,B 0,C 180,E1 -1794.441,E2 -1794.441} C_VEL
LIN {X 0,Y 580.345,Z 512.19,A -85,B 0,C 180,E1 -1797.224,E2 -1797.224} C_VEL
LIN {X 0,Y 580.359,Z 512.194,A -85,B 0,C 180,E1 -1800,E2 -1800} C_VEL
LIN {X 0,Y 580.345,Z 512.188,A -85,B 0,C 180,E1 -1802.777,E2 -1802.777} C_VEL
LIN {X 0,Y 580.327,Z 512.196,A -85,B 0,C 180,E1 -1805.56,E2 -1805.56} C_VEL
LIN {X 0,Y 580.333,Z 512.193,A -85,B 0,C 180,E1 -1808.356,E2 -1808.356} C_VEL
LIN {X 0,Y 580.308,Z 512.194,A -85,B 0,C 180,E1 -1811.191,E2 -1811.191} C_VEL
LIN {X 0,Y 580.332,Z 512.2,A -85,B 0,C 180,E1 -1814.017,E2 -1814.017} C_VEL
LIN {X 0,Y 580.32,Z 512.191,A -85,B 0,C 180,E1 -1816.914,E2 -1816.914} C_VEL
LIN {X 0,Y 580.294,Z 512.202,A -85,B 0,C 180,E1 -1819.823,E2 -1819.823} C_VEL
LIN {X 0,Y 580.28,Z 512.207,A -85,B 0,C 180,E1 -1822.053,E2 -1822.053} C_VEL
LIN {X 0,Y 580.313,Z 512.192,A -85,B 0,C 180,E1 -1825.08,E2 -1825.08} C_VEL
LIN {X 0,Y 580.303,Z 512.203,A -85,B 0,C 180,E1 -1828.186,E2 -1828.186} C_VEL
LIN {X 0,Y 580.29,Z 512.197,A -85,B 0,C 180,E1 -1830.694,E2 -1830.694} C_VEL
LIN {X 0,Y 580.29,Z 512.195,A -85,B 0,C 180,E1 -1833.313,E2 -1833.313} C_VEL
LIN {X 0,Y 580.271,Z 512.201,A -85,B 0,C 180,E1 -1835.759,E2 -1835.759} C_VEL
LIN {X 0,Y 580.294,Z 512.204,A -85,B 0,C 180,E1 -1838.146,E2 -1838.146} C_VEL
LIN {X 0,Y 580.303,Z 512.195,A -85,B 0,C 180,E1 -1840.843,E2 -1840.843} C_VEL
LIN {X 0,Y 580.249,Z 512.202,A -85,B 0,C 180,E1 -1843.661,E2 -1843.661} C_VEL
LIN {X 0,Y 580.29,Z 512.201,A -85,B 0,C 180,E1 -1846.608,E2 -1846.608} C_VEL
LIN {X 0,Y 580.304,Z 512.194,A -85,B 0,C 180,E1 -1849.156,E2 -1849.156} C_VEL
LIN {X 0,Y 580.295,Z 512.198,A -85,B 0,C 180,E1 -1851.927,E2 -1851.927} C_VEL
LIN {X 0,Y 580.258,Z 512.209,A -85,B 0,C 180,E1 -1854.452,E2 -1854.452} C_VEL
LIN {X 0,Y 580.297,Z 512.196,A -85,B 0,C 180,E1 -1856.975,E2 -1856.975} C_VEL
LIN {X 0,Y 580.302,Z 512.194,A -85,B 0,C 180,E1 -1859.425,E2 -1859.425} C_VEL
LIN {X 0,Y 580.303,Z 512.199,A -85,B 0,C 180,E1 -1862.141,E2 -1862.141} C_VEL
LIN {X 0,Y 580.328,Z 512.193,A -85,B 0,C 180,E1 -1865.269,E2 -1865.269} C_VEL
LIN {X 0,Y 580.321,Z 512.358,A -85,B 0,C 180,E1 -1867.105,E2 -1867.105} C_VEL
LIN {X 0,Y 580.917,Z 516.755,A -85,B 0,C 180,E1 -1867.785,E2 -1867.785} C_VEL
LIN {X 0,Y 580.703,Z 536.853,A -85,B 0,C 180,E1 -1870.735,E2 -1870.735} C_VEL
LIN {X 0,Y 580.523,Z 555.794,A -85,B 0,C 180,E1 -1873.47,E2 -1873.47} C_VEL
LIN {X 0,Y 580.393,Z 576.069,A -85,B 0,C 180,E1 -1876.341,E2 -1876.341} C_VEL
LIN {X 0,Y 580.961,Z 581.435,A -85,B 0,C 180,E1 -1876.422,E2 -1876.422} C_VEL
LIN {X 0,Y 580.808,Z 683.899,A -85,B 0,C 180,E1 -1877.707,E2 -1877.707} C_VEL
LIN {X 0,Y 580.74,Z 697.188,A -85,B 0,C 180,E1 -1878.016,E2 -1878.016} C_VEL
LIN {X 0,Y 580.654,Z 710.47,A -85,B 0,C 180,E1 -1878.479,E2 -1878.479} C_VEL
LIN {X 0,Y 580.546,Z 721.614,A -85,B 0,C 180,E1 -1879.007,E2 -1879.007} C_VEL
LIN {X 0,Y 580.427,Z 733.189,A -85,B 0,C 180,E1 -1879.711,E2 -1879.711} C_VEL
LIN {X 0,Y 580.341,Z 743.587,A -85,B 0,C 180,E1 -1880.502,E2 -1880.502} C_VEL
LIN {X 0,Y 580.267,Z 752.103,A -85,B 0,C 180,E1 -1881.291,E2 -1881.291} C_VEL
LIN {X 0,Y 580.222,Z 759.953,A -85,B 0,C 180,E1 -1882.167,E2 -1882.167} C_VEL
LIN {X 0,Y 580.155,Z 767.646,A -85,B 0,C 180,E1 -1883.221,E2 -1883.221} C_VEL
LIN {X 0,Y 580.139,Z 774.675,A -85,B 0,C 180,E1 -1884.438,E2 -1884.438} C_VEL
LIN {X 0,Y 580.108,Z 779.368,A -85,B 0,C 180,E1 -1885.482,E2 -1885.482} C_VEL
LIN {X 0,Y 580.123,Z 782.954,A -85,B 0,C 180,E1 -1886.526,E2 -1886.526} C_VEL
LIN {X 0,Y 580.043,Z 784.806,A -85,B 0,C 180,E1 -1887.221,E2 -1887.221} C_VEL
LIN {X 0,Y 580.038,Z 786.198,A -85,B 0,C 180,E1 -1887.916,E2 -1887.916} C_VEL
LIN {X 0,Y 580.04,Z 787.784,A -85,B 0,C 180,E1 -1889.305,E2 -1889.305} C_VEL
LIN {X 0,Y 580.037,Z 788,A -85,B 0,C 180,E1 -1889.999,E2 -1889.999} C_VEL
LIN {X 0,Y 580.047,Z 787.187,A -85,B 0,C 180,E1 -1891.388,E2 -1891.388} C_VEL
LIN {X 0,Y 580.038,Z 786.202,A -85,B 0,C 180,E1 -1892.082,E2 -1892.082} C_VEL
LIN {X 0,Y 580.043,Z 784.812,A -85,B 0,C 180,E1 -1892.777,E2 -1892.777} C_VEL
LIN {X 0,Y 580.109,Z 781.899,A -85,B 0,C 180,E1 -1893.82,E2 -1893.82} C_VEL
LIN {X 0,Y 580.054,Z 777.953,A -85,B 0,C 180,E1 -1894.864,E2 -1894.864} C_VEL
LIN {X 0,Y 580.139,Z 771.883,A -85,B 0,C 180,E1 -1896.084,E2 -1896.084} C_VEL
LIN {X 0,Y 580.184,Z 765.244,A -85,B 0,C 180,E1 -1897.131,E2 -1897.131} C_VEL
LIN {X 0,Y 580.25,Z 756.999,A -85,B 0,C 180,E1 -1898.181,E2 -1898.181} C_VEL
LIN {X 0,Y 580.307,Z 748.549,A -85,B 0,C 180,E1 -1899.057,E2 -1899.057} C_VEL
LIN {X 0,Y 580.414,Z 738.11,A -85,B 0,C 180,E1 -1899.935,E2 -1899.935} C_VEL
LIN {X 0,Y 580.521,Z 727.775,A -85,B 0,C 180,E1 -1900.638,E2 -1900.638} C_VEL
LIN {X 0,Y 580.596,Z 716.252,A -85,B 0,C 180,E1 -1901.264,E2 -1901.264} C_VEL
LIN {X 0,Y 580.664,Z 703.504,A -85,B 0,C 180,E1 -1901.784,E2 -1901.784} C_VEL
LIN {X 0,Y 580.765,Z 690.481,A -85,B 0,C 180,E1 -1902.159,E2 -1902.159} C_VEL
LIN {X 0,Y 580.826,Z 678.165,A -85,B 0,C 180,E1 -1902.379,E2 -1902.379} C_VEL
LIN {X 0,Y 580.789,Z 578.592,A -85,B 0,C 180,E1 -1903.618,E2 -1903.618} C_VEL
LIN {X 0,Y 580.382,Z 575.8,A -85,B 0,C 180,E1 -1903.679,E2 -1903.679} C_VEL
LIN {X 0,Y 580.521,Z 555.809,A -85,B 0,C 180,E1 -1906.528,E2 -1906.528} C_VEL
LIN {X 0,Y 580.703,Z 536.853,A -85,B 0,C 180,E1 -1909.265,E2 -1909.265} C_VEL
LIN {X 0,Y 580.918,Z 516.77,A -85,B 0,C 180,E1 -1912.213,E2 -1912.213} C_VEL
LIN {X 0,Y 580.283,Z 512.205,A -85,B 0,C 180,E1 -1912.926,E2 -1912.926} C_VEL
LIN {X 0,Y 580.305,Z 512.2,A -85,B 0,C 180,E1 -1915.078,E2 -1915.078} C_VEL
LIN {X 0,Y 580.299,Z 512.197,A -85,B 0,C 180,E1 -1918.184,E2 -1918.184} C_VEL
LIN {X 0,Y 580.291,Z 512.197,A -85,B 0,C 180,E1 -1920.695,E2 -1920.695} C_VEL
LIN {X 0,Y 580.302,Z 512.202,A -85,B 0,C 180,E1 -1923.316,E2 -1923.316} C_VEL
LIN {X 0,Y 580.272,Z 512.204,A -85,B 0,C 180,E1 -1925.759,E2 -1925.759} C_VEL
LIN {X 0,Y 580.286,Z 512.198,A -85,B 0,C 180,E1 -1928.145,E2 -1928.145} C_VEL
LIN {X 0,Y 580.297,Z 512.197,A -85,B 0,C 180,E1 -1930.842,E2 -1930.842} C_VEL
LIN {X 0,Y 580.283,Z 512.204,A -85,B 0,C 180,E1 -1933.656,E2 -1933.656} C_VEL
LIN {X 0,Y 580.27,Z 512.199,A -85,B 0,C 180,E1 -1936.608,E2 -1936.608} C_VEL
LIN {X 0,Y 580.294,Z 512.201,A -85,B 0,C 180,E1 -1939.156,E2 -1939.156} C_VEL
LIN {X 0,Y 580.283,Z 512.199,A -85,B 0,C 180,E1 -1941.926,E2 -1941.926} C_VEL
LIN {X 0,Y 580.302,Z 512.194,A -85,B 0,C 180,E1 -1944.456,E2 -1944.456} C_VEL
LIN {X 0,Y 580.285,Z 512.199,A -85,B 0,C 180,E1 -1946.974,E2 -1946.974} C_VEL
LIN {X 0,Y 580.301,Z 512.204,A -85,B 0,C 180,E1 -1949.425,E2 -1949.425} C_VEL
LIN {X 0,Y 580.311,Z 512.193,A -85,B 0,C 180,E1 -1952.136,E2 -1952.136} C_VEL
LIN {X 0,Y 580.301,Z 512.197,A -85,B 0,C 180,E1 -1954.92,E2 -1954.92} C_VEL
LIN {X 0,Y 580.266,Z 512.201,A -85,B 0,C 180,E1 -1957.947,E2 -1957.947} C_VEL
LIN {X 0,Y 580.308,Z 512.195,A -85,B 0,C 180,E1 -1960.913,E2 -1960.913} C_VEL
LIN {X 0,Y 580.273,Z 512.201,A -85,B 0,C 180,E1 -1963.825,E2 -1963.825} C_VEL
LIN {X 0,Y 580.316,Z 512.195,A -85,B 0,C 180,E1 -1965.982,E2 -1965.982} C_VEL
LIN {X 0,Y 580.321,Z 512.193,A -85,B 0,C 180,E1 -1968.827,E2 -1968.827} C_VEL
LIN {X 0,Y 580.327,Z 512.197,A -85,B 0,C 180,E1 -1971.644,E2 -1971.644} C_VEL
LIN {X 0,Y 580.317,Z 512.192,A -85,B 0,C 180,E1 -1974.44,E2 -1974.44} C_VEL
LIN {X 0,Y 580.341,Z 512.196,A -85,B 0,C 180,E1 -1977.223,E2 -1977.223} C_VEL
LIN {X 0,Y 580.342,Z 512.191,A -85,B 0,C 180,E1 -1980,E2 -1980} C_VEL
LIN {X 0,Y 580.339,Z 512.191,A -85,B 0,C 180,E1 -1982.776,E2 -1982.776} C_VEL
LIN {X 0,Y 580.316,Z 512.2,A -85,B 0,C 180,E1 -1985.559,E2 -1985.559} C_VEL
LIN {X 0,Y 580.326,Z 512.191,A -85,B 0,C 180,E1 -1988.356,E2 -1988.356} C_VEL
LIN {X 0,Y 580.321,Z 512.199,A -85,B 0,C 180,E1 -1991.208,E2 -1991.208} C_VEL
LIN {X 0,Y 580.315,Z 512.195,A -85,B 0,C 180,E1 -1994.017,E2 -1994.017} C_VEL
LIN {X 0,Y 580.303,Z 512.198,A -85,B 0,C 180,E1 -1996.915,E2 -1996.915} C_VEL
LIN {X 0,Y 580.298,Z 512.199,A -85,B 0,C 180,E1 -1999.822,E2 -1999.822} C_VEL
LIN {X 0,Y 580.277,Z 512.206,A -85,B 0,C 180,E1 -2001.344,E2 -2001.344} C_VEL
LIN {X 0,Y 579.58,Z 512.288,A -85,B 0,C 180,E1 -2001.923,E2 -2001.923} C_VEL
LIN {X 0,Y 576.702,Z 512.646,A -85,B 0,C 180,E1 -2002.863,E2 -2002.863} C_VEL
LIN {X 0,Y 574.306,Z 512.948,A -85,B 0,C 180,E1 -2003.619,E2 -2003.619} C_VEL
LIN {X 0,Y 573.307,Z 513.067,A -85,B 0,C 180,E1 -2004.203,E2 -2004.203} C_VEL
LIN {X 0,Y 573.24,Z 513.075,A -85,B 0,C 180,E1 -2004.401,E2 -2004.401} C_VEL
LIN {X 0,Y 573.257,Z 513.077,A -85,B 0,C 180,E1 -2006.975,E2 -2006.975} C_VEL
LIN {X 0,Y 573.318,Z 513.167,A -85,B 0,C 180,E1 -2010.273,E2 -2010.273} C_VEL
LIN {X 0,Y 573.527,Z 519.397,A -85,B 0,C 180,E1 -2011.385,E2 -2011.385} C_VEL
LIN {X 0,Y 573.367,Z 536.177,A -85,B 0,C 180,E1 -2014.321,E2 -2014.321} C_VEL
LIN {X 0,Y 573.269,Z 547.096,A -85,B 0,C 180,E1 -2016.21,E2 -2016.21} C_VEL
LIN {X 0,Y 574.057,Z 553.745,A -85,B 0,C 180,E1 -2016.329,E2 -2016.329} C_VEL
LIN {X 0,Y 573.878,Z 654.457,A -85,B 0,C 180,E1 -2017.612,E2 -2017.612} C_VEL
LIN {X 0,Y 573.771,Z 667.47,A -85,B 0,C 180,E1 -2017.922,E2 -2017.922} C_VEL
LIN {X 0,Y 573.691,Z 680.18,A -85,B 0,C 180,E1 -2018.371,E2 -2018.371} C_VEL
LIN {X 0,Y 573.588,Z 692.278,A -85,B 0,C 180,E1 -2018.955,E2 -2018.955} C_VEL
LIN {X 0,Y 573.421,Z 704.306,A -85,B 0,C 180,E1 -2019.706,E2 -2019.706} C_VEL
LIN {X 0,Y 573.316,Z 714.814,A -85,B 0,C 180,E1 -2020.535,E2 -2020.535} C_VEL
LIN {X 0,Y 573.219,Z 724.265,A -85,B 0,C 180,E1 -2021.457,E2 -2021.457} C_VEL
LIN {X 0,Y 573.106,Z 732.261,A -85,B 0,C 180,E1 -2022.412,E2 -2022.412} C_VEL
LIN {X 0,Y 573.067,Z 738.88,A -85,B 0,C 180,E1 -2023.375,E2 -2023.375} C_VEL
LIN {X 0,Y 573.044,Z 744.37,A -85,B 0,C 180,E1 -2024.352,E2 -2024.352} C_VEL
LIN {X 0,Y 573.008,Z 748.873,A -85,B 0,C 180,E1 -2025.346,E2 -2025.346} C_VEL
LIN {X 0,Y 572.964,Z 753.218,A -85,B 0,C 180,E1 -2026.617,E2 -2026.617} C_VEL
LIN {X 0,Y 572.984,Z 755.531,A -85,B 0,C 180,E1 -2027.578,E2 -2027.578} C_VEL
LIN {X 0,Y 572.939,Z 757.052,A -85,B 0,C 180,E1 -2028.519,E2 -2028.519} C_VEL
LIN {X 0,Y 572.932,Z 757.885,A -85,B 0,C 180,E1 -2029.511,E2 -2029.511} C_VEL
LIN {X 0,Y 572.915,Z 757.873,A -85,B 0,C 180,E1 -2030.608,E2 -2030.608} C_VEL
LIN {X 0,Y 572.922,Z 756.863,A -85,B 0,C 180,E1 -2031.728,E2 -2031.728} C_VEL
LIN {X 0,Y 572.97,Z 754.311,A -85,B 0,C 180,E1 -2033.058,E2 -2033.058} C_VEL
LIN {X 0,Y 573.027,Z 750.114,A -85,B 0,C 180,E1 -2034.427,E2 -2034.427} C_VEL
LIN {X 0,Y 572.998,Z 744.796,A -85,B 0,C 180,E1 -2035.654,E2 -2035.654} C_VEL
LIN {X 0,Y 573.077,Z 738.869,A -85,B 0,C 180,E1 -2036.717,E2 -2036.717} C_VEL
LIN {X 0,Y 573.119,Z 731.386,A -85,B 0,C 180,E1 -2037.792,E2 -2037.792} C_VEL
LIN {X 0,Y 573.255,Z 722.644,A -85,B 0,C 180,E1 -2038.805,E2 -2038.805} C_VEL
LIN {X 0,Y 573.36,Z 712.763,A -85,B 0,C 180,E1 -2039.73,E2 -2039.73} C_VEL
LIN {X 0,Y 573.435,Z 701.88,A -85,B 0,C 180,E1 -2040.551,E2 -2040.551} C_VEL
LIN {X 0,Y 573.582,Z 690.048,A -85,B 0,C 180,E1 -2041.256,E2 -2041.256} C_VEL
LIN {X 0,Y 573.691,Z 677.174,A -85,B 0,C 180,E1 -2041.839,E2 -2041.839} C_VEL
LIN {X 0,Y 573.786,Z 664.184,A -85,B 0,C 180,E1 -2042.263,E2 -2042.263} C_VEL
LIN {X 0,Y 573.875,Z 650.647,A -85,B 0,C 180,E1 -2042.539,E2 -2042.539} C_VEL
LIN {X 0,Y 573.998,Z 551.463,A -85,B 0,C 180,E1 -2043.791,E2 -2043.791} C_VEL
LIN {X 0,Y 573.286,Z 547.26,A -85,B 0,C 180,E1 -2043.862,E2 -2043.862} C_VEL
LIN {X 0,Y 573.388,Z 531.861,A -85,B 0,C 180,E1 -2046.52,E2 -2046.52} C_VEL
LIN {X 0,Y 573.549,Z 515.614,A -85,B 0,C 180,E1 -2049.374,E2 -2049.374} C_VEL
LIN {X 0,Y 573.252,Z 513.079,A -85,B 0,C 180,E1 -2049.878,E2 -2049.878} C_VEL
LIN {X 0,Y 573.256,Z 513.079,A -85,B 0,C 180,E1 -2052.99,E2 -2052.99} C_VEL
LIN {X 0,Y 573.27,Z 513.07,A -85,B 0,C 180,E1 -2055.808,E2 -2055.808} C_VEL
LIN {X 0,Y 573.258,Z 513.081,A -85,B 0,C 180,E1 -2058.746,E2 -2058.746} C_VEL
LIN {X 0,Y 573.282,Z 513.069,A -85,B 0,C 180,E1 -2061.542,E2 -2061.542} C_VEL
LIN {X 0,Y 573.296,Z 513.069,A -85,B 0,C 180,E1 -2064.373,E2 -2064.373} C_VEL
LIN {X 0,Y 573.312,Z 513.064,A -85,B 0,C 180,E1 -2067.893,E2 -2067.893} C_VEL
LIN {X 0,Y 573.331,Z 513.069,A -85,B 0,C 180,E1 -2070.703,E2 -2070.703} C_VEL
LIN {X 0,Y 573.304,Z 513.074,A -85,B 0,C 180,E1 -2072.812,E2 -2072.812} C_VEL
LIN {X 0,Y 573.293,Z 513.068,A -85,B 0,C 180,E1 -2075.629,E2 -2075.629} C_VEL
LIN {X 0,Y 573.282,Z 513.07,A -85,B 0,C 180,E1 -2078.46,E2 -2078.46} C_VEL
LIN {X 0,Y 573.271,Z 513.075,A -85,B 0,C 180,E1 -2081.313,E2 -2081.313} C_VEL
LIN {X 0,Y 573.281,Z 513.07,A -85,B 0,C 180,E1 -2084.425,E2 -2084.425} C_VEL
LIN {X 0,Y 573.258,Z 513.082,A -85,B 0,C 180,E1 -2087.113,E2 -2087.113} C_VEL
LIN {X 0,Y 573.251,Z 513.072,A -85,B 0,C 180,E1 -2090.078,E2 -2090.078} C_VEL
LIN {X 0,Y 573.235,Z 513.084,A -85,B 0,C 180,E1 -2093.1,E2 -2093.1} C_VEL
LIN {X 0,Y 573.253,Z 513.078,A -85,B 0,C 180,E1 -2095.411,E2 -2095.411} C_VEL
LIN {X 0,Y 573.251,Z 513.072,A -85,B 0,C 180,E1 -2098.03,E2 -2098.03} C_VEL
LIN {X 0,Y 573.24,Z 513.078,A -85,B 0,C 180,E1 -2100.885,E2 -2100.885} C_VEL
LIN {X 0,Y 573.264,Z 513.076,A -85,B 0,C 180,E1 -2103.525,E2 -2103.525} C_VEL
LIN {X 0,Y 573.216,Z 513.077,A -85,B 0,C 180,E1 -2106.052,E2 -2106.052} C_VEL
LIN {X 0,Y 573.25,Z 513.074,A -85,B 0,C 180,E1 -2108.702,E2 -2108.702} C_VEL
LIN {X 0,Y 573.256,Z 513.078,A -85,B 0,C 180,E1 -2111.596,E2 -2111.596} C_VEL
LIN {X 0,Y 573.242,Z 513.073,A -85,B 0,C 180,E1 -2114.334,E2 -2114.334} C_VEL
LIN {X 0,Y 573.242,Z 513.083,A -85,B 0,C 180,E1 -2117.359,E2 -2117.359} C_VEL
LIN {X 0,Y 573.25,Z 513.072,A -85,B 0,C 180,E1 -2120.394,E2 -2120.394} C_VEL
LIN {X 0,Y 573.254,Z 513.076,A -85,B 0,C 180,E1 -2123.078,E2 -2123.078} C_VEL
LIN {X 0,Y 573.275,Z 513.076,A -85,B 0,C 180,E1 -2125.672,E2 -2125.672} C_VEL
LIN {X 0,Y 573.244,Z 513.074,A -85,B 0,C 180,E1 -2128.185,E2 -2128.185} C_VEL
LIN {X 0,Y 573.269,Z 513.07,A -85,B 0,C 180,E1 -2130.635,E2 -2130.635} C_VEL
LIN {X 0,Y 573.242,Z 513.083,A -85,B 0,C 180,E1 -2133.508,E2 -2133.508} C_VEL
LIN {X 0,Y 573.232,Z 513.077,A -85,B 0,C 180,E1 -2136.135,E2 -2136.135} C_VEL
LIN {X 0,Y 573.255,Z 513.075,A -85,B 0,C 180,E1 -2139.174,E2 -2139.174} C_VEL
LIN {X 0,Y 573.226,Z 513.082,A -85,B 0,C 180,E1 -2141.412,E2 -2141.412} C_VEL
LIN {X 0,Y 573.256,Z 513.082,A -85,B 0,C 180,E1 -2143.622,E2 -2143.622} C_VEL
LIN {X 0,Y 573.278,Z 513.077,A -85,B 0,C 180,E1 -2145.808,E2 -2145.808} C_VEL
LIN {X 0,Y 573.269,Z 513.07,A -85,B 0,C 180,E1 -2148.746,E2 -2148.746} C_VEL
LIN {X 0,Y 573.289,Z 513.074,A -85,B 0,C 180,E1 -2151.541,E2 -2151.541} C_VEL
LIN {X 0,Y 573.292,Z 513.069,A -85,B 0,C 180,E1 -2154.372,E2 -2154.372} C_VEL
LIN {X 0,Y 573.314,Z 513.073,A -85,B 0,C 180,E1 -2157.893,E2 -2157.893} C_VEL
LIN {X 0,Y 573.337,Z 513.061,A -85,B 0,C 180,E1 -2160.703,E2 -2160.703} C_VEL
LIN {X 0,Y 573.311,Z 513.064,A -85,B 0,C 180,E1 -2162.811,E2 -2162.811} C_VEL
LIN {X 0,Y 573.295,Z 513.073,A -85,B 0,C 180,E1 -2165.628,E2 -2165.628} C_VEL
LIN {X 0,Y 573.289,Z 513.07,A -85,B 0,C 180,E1 -2168.46,E2 -2168.46} C_VEL
LIN {X 0,Y 573.279,Z 513.07,A -85,B 0,C 180,E1 -2171.312,E2 -2171.312} C_VEL
LIN {X 0,Y 573.289,Z 513.071,A -85,B 0,C 180,E1 -2174.424,E2 -2174.424} C_VEL
LIN {X 0,Y 573.266,Z 513.07,A -85,B 0,C 180,E1 -2177.112,E2 -2177.112} C_VEL
LIN {X 0,Y 573.249,Z 513.082,A -85,B 0,C 180,E1 -2180.077,E2 -2180.077} C_VEL
LIN {X 0,Y 573.242,Z 513.079,A -85,B 0,C 180,E1 -2182.338,E2 -2182.338} C_VEL
LIN {X 0,Y 573.26,Z 513.072,A -85,B 0,C 180,E1 -2185.41,E2 -2185.41} C_VEL
LIN {X 0,Y 573.243,Z 513.076,A -85,B 0,C 180,E1 -2188.565,E2 -2188.565} C_VEL
LIN {X 0,Y 573.232,Z 513.075,A -85,B 0,C 180,E1 -2190.993,E2 -2190.993} C_VEL
LIN {X 0,Y 573.248,Z 513.074,A -85,B 0,C 180,E1 -2193.521,E2 -2193.521} C_VEL
LIN {X 0,Y 573.247,Z 513.081,A -85,B 0,C 180,E1 -2196.05,E2 -2196.05} C_VEL
LIN {X 0,Y 573.249,Z 513.075,A -85,B 0,C 180,E1 -2198.701,E2 -2198.701} C_VEL
LIN {X 0,Y 573.236,Z 513.075,A -85,B 0,C 180,E1 -2201.593,E2 -2201.593} C_VEL
LIN {X 0,Y 573.219,Z 513.08,A -85,B 0,C 180,E1 -2204.673,E2 -2204.673} C_VEL
LIN {X 0,Y 573.25,Z 513.072,A -85,B 0,C 180,E1 -2207.358,E2 -2207.358} C_VEL
LIN {X 0,Y 573.246,Z 513.083,A -85,B 0,C 180,E1 -2210.392,E2 -2210.392} C_VEL
LIN {X 0,Y 573.258,Z 513.072,A -85,B 0,C 180,E1 -2213.077,E2 -2213.077} C_VEL
LIN {X 0,Y 573.273,Z 513.07,A -85,B 0,C 180,E1 -2215.671,E2 -2215.671} C_VEL
LIN {X 0,Y 573.247,Z 513.079,A -85,B 0,C 180,E1 -2218.184,E2 -2218.184} C_VEL
LIN {X 0,Y 573.27,Z 513.077,A -85,B 0,C 180,E1 -2220.634,E2 -2220.634} C_VEL
LIN {X 0,Y 573.256,Z 513.074,A -85,B 0,C 180,E1 -2223.023,E2 -2223.023} C_VEL
LIN {X 0,Y 573.282,Z 513.071,A -85,B 0,C 180,E1 -2225.366,E2 -2225.366} C_VEL
LIN {X 0,Y 573.258,Z 513.212,A -85,B 0,C 180,E1 -2226.936,E2 -2226.936} C_VEL
LIN {X 0,Y 574.003,Z 518.015,A -85,B 0,C 180,E1 -2227.693,E2 -2227.693} C_VEL
LIN {X 0,Y 573.754,Z 538.164,A -85,B 0,C 180,E1 -2230.686,E2 -2230.686} C_VEL
LIN {X 0,Y 573.545,Z 557.099,A -85,B 0,C 180,E1 -2233.453,E2 -2233.453} C_VEL
LIN {X 0,Y 573.4,Z 576.069,A -85,B 0,C 180,E1 -2236.171,E2 -2236.171} C_VEL
LIN {X 0,Y 574.059,Z 581.435,A -85,B 0,C 180,E1 -2236.255,E2 -2236.255} C_VEL
LIN {X 0,Y 573.874,Z 683.899,A -85,B 0,C 180,E1 -2237.556,E2 -2237.556} C_VEL
LIN {X 0,Y 573.794,Z 697.188,A -85,B 0,C 180,E1 -2237.869,E2 -2237.869} C_VEL
LIN {X 0,Y 573.712,Z 709.35,A -85,B 0,C 180,E1 -2238.293,E2 -2238.293} C_VEL
LIN {X 0,Y 573.592,Z 720.561,A -85,B 0,C 180,E1 -2238.816,E2 -2238.816} C_VEL
LIN {X 0,Y 573.471,Z 731.898,A -85,B 0,C 180,E1 -2239.496,E2 -2239.496} C_VEL
LIN {X 0,Y 573.343,Z 742.529,A -85,B 0,C 180,E1 -2240.296,E2 -2240.296} C_VEL
LIN {X 0,Y 573.239,Z 752.103,A -85,B 0,C 180,E1 -2241.184,E2 -2241.184} C_VEL
LIN {X 0,Y 573.162,Z 759.953,A -85,B 0,C 180,E1 -2242.07,E2 -2242.07} C_VEL
LIN {X 0,Y 573.074,Z 767.95,A -85,B 0,C 180,E1 -2243.185,E2 -2243.185} C_VEL
LIN {X 0,Y 573.07,Z 774.675,A -85,B 0,C 180,E1 -2244.369,E2 -2244.369} C_VEL
LIN {X 0,Y 573.029,Z 779.368,A -85,B 0,C 180,E1 -2245.427,E2 -2245.427} C_VEL
LIN {X 0,Y 573.023,Z 782.954,A -85,B 0,C 180,E1 -2246.483,E2 -2246.483} C_VEL
LIN {X 0,Y 572.959,Z 784.806,A -85,B 0,C 180,E1 -2247.187,E2 -2247.187} C_VEL
LIN {X 0,Y 572.937,Z 786.197,A -85,B 0,C 180,E1 -2247.89,E2 -2247.89} C_VEL
LIN {X 0,Y 572.941,Z 787.784,A -85,B 0,C 180,E1 -2249.296,E2 -2249.296} C_VEL
LIN {X 0,Y 572.938,Z 788,A -85,B 0,C 180,E1 -2249.999,E2 -2249.999} C_VEL
LIN {X 0,Y 572.946,Z 787.187,A -85,B 0,C 180,E1 -2251.405,E2 -2251.405} C_VEL
LIN {X 0,Y 572.937,Z 786.202,A -85,B 0,C 180,E1 -2252.108,E2 -2252.108} C_VEL
LIN {X 0,Y 572.959,Z 784.812,A -85,B 0,C 180,E1 -2252.811,E2 -2252.811} C_VEL
LIN {X 0,Y 573.014,Z 781.899,A -85,B 0,C 180,E1 -2253.867,E2 -2253.867} C_VEL
LIN {X 0,Y 572.963,Z 777.953,A -85,B 0,C 180,E1 -2254.925,E2 -2254.925} C_VEL
LIN {X 0,Y 573.064,Z 771.883,A -85,B 0,C 180,E1 -2256.159,E2 -2256.159} C_VEL
LIN {X 0,Y 573.119,Z 765.245,A -85,B 0,C 180,E1 -2257.22,E2 -2257.22} C_VEL
LIN {X 0,Y 573.2,Z 756.999,A -85,B 0,C 180,E1 -2258.282,E2 -2258.282} C_VEL
LIN {X 0,Y 573.286,Z 748.55,A -85,B 0,C 180,E1 -2259.169,E2 -2259.169} C_VEL
LIN {X 0,Y 573.42,Z 738.111,A -85,B 0,C 180,E1 -2260.057,E2 -2260.057} C_VEL
LIN {X 0,Y 573.545,Z 727.79,A -85,B 0,C 180,E1 -2260.768,E2 -2260.768} C_VEL
LIN {X 0,Y 573.627,Z 716.61,A -85,B 0,C 180,E1 -2261.384,E2 -2261.384} C_VEL
LIN {X 0,Y 573.698,Z 704.8,A -85,B 0,C 180,E1 -2261.884,E2 -2261.884} C_VEL
LIN {X 0,Y 573.848,Z 691.395,A -85,B 0,C 180,E1 -2262.285,E2 -2262.285} C_VEL
LIN {X 0,Y 573.904,Z 678.165,A -85,B 0,C 180,E1 -2262.531,E2 -2262.531} C_VEL
LIN {X 0,Y 573.958,Z 579.81,A -85,B 0,C 180,E1 -2263.768,E2 -2263.768} C_VEL
LIN {X 0,Y 573.393,Z 575.8,A -85,B 0,C 180,E1 -2263.849,E2 -2263.849} C_VEL
LIN {X 0,Y 573.542,Z 555.897,A -85,B 0,C 180,E1 -2266.722,E2 -2266.722} C_VEL
LIN {X 0,Y 573.745,Z 537.561,A -85,B 0,C 180,E1 -2269.403,E2 -2269.403} C_VEL
LIN {X 0,Y 574.014,Z 518.029,A -85,B 0,C 180,E1 -2272.305,E2 -2272.305} C_VEL
LIN {X 0,Y 573.234,Z 513.085,A -85,B 0,C 180,E1 -2273.098,E2 -2273.098} C_VEL
LIN {X 0,Y 573.253,Z 513.083,A -85,B 0,C 180,E1 -2275.409,E2 -2275.409} C_VEL
LIN {X 0,Y 573.251,Z 513.076,A -85,B 0,C 180,E1 -2278.028,E2 -2278.028} C_VEL
LIN {X 0,Y 573.237,Z 513.077,A -85,B 0,C 180,E1 -2280.883,E2 -2280.883} C_VEL
LIN {X 0,Y 573.259,Z 513.081,A -85,B 0,C 180,E1 -2283.523,E2 -2283.523} C_VEL
LIN {X 0,Y 573.241,Z 513.076,A -85,B 0,C 180,E1 -2286.048,E2 -2286.048} C_VEL
LIN {X 0,Y 573.245,Z 513.074,A -85,B 0,C 180,E1 -2288.7,E2 -2288.7} C_VEL
LIN {X 0,Y 573.25,Z 513.081,A -85,B 0,C 180,E1 -2291.595,E2 -2291.595} C_VEL
LIN {X 0,Y 573.233,Z 513.075,A -85,B 0,C 180,E1 -2294.332,E2 -2294.332} C_VEL
LIN {X 0,Y 573.233,Z 513.084,A -85,B 0,C 180,E1 -2297.357,E2 -2297.357} C_VEL
